KUKA KRL program: MyProgram_312().src

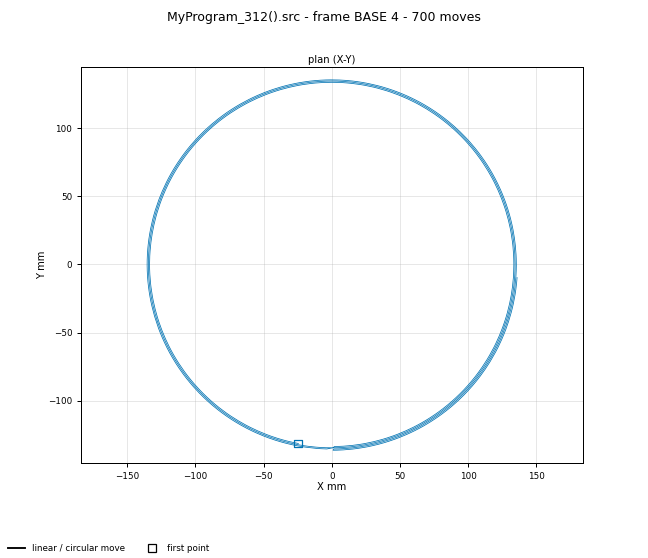
[picture p0: tool path of MyProgram_312().src in frame BASE 4, 700 of 700 moves have a stored position in this frame; points joined in program order, loops and branches not executed]
&ACCESS RVP
&REL 1
&PARAM TEMPLATE = C:\KRC\Roboter\Template\vorgabe
&PARAM EDITMASK = *
DEF MyProgram_312()
; ---- Setting reference (Base) ----
$BASE = BASE_DATA[4]

; --------------------------
; ---- Setting tool (TCP) ----
$TOOL = TOOL_DATA[3]
; --------------------------

$VEL.CP = VEL_APROX_PRINT
Startdeposition()
$VEL.CP = VEL_PRINT
LIN {X -24.4618,Y -131.3769,Z 183,A -96.3174,B 4.4526,C 0.3571,E1 4.4393,E2 188.8666} C_DIS
LIN {X -27.6736,Y -130.7376,Z 183,A -97.6133,B 4.4528,C 0.3555,E1 4.4357,E2 190.1492} C_DIS
LIN {X -30.5793,Y -130.0897,Z 183,A -99.1035,B 4.4527,C 0.3569,E1 4.4316,E2 191.6668} C_DIS
LIN {X -33.6463,Y -129.3306,Z 183,A -100.4108,B 4.4527,C 0.3557,E1 4.4281,E2 192.9686} C_DIS
LIN {X -36.9217,Y -128.4331,Z 183,A -101.7714,B 4.4529,C 0.3539,E1 4.4245,E2 194.3175} C_DIS
LIN {X -40.1243,Y -127.4684,Z 183,A -103.4209,B 4.4529,C 0.3548,E1 4.42,E2 195.9945} C_DIS
LIN {X -44.4742,Y -126.0175,Z 183,A -105.417,B 4.4529,C 0.3535,E1 4.4147,E2 197.9948} C_DIS
LIN {X -48.1013,Y -124.6763,Z 183,A -106.9374,B 4.4531,C 0.3508,E1 4.4108,E2 199.4981} C_DIS
LIN {X -51.1439,Y -123.4595,Z 183,A -108.3574,B 4.4532,C 0.3496,E1 4.4071,E2 200.9202} C_DIS
LIN {X -54.1545,Y -122.1691,Z 183,A -109.7774,B 4.4533,C 0.3483,E1 4.4034,E2 202.3424} C_DIS
LIN {X -57.1353,Y -120.804,Z 183,A -111.0888,B 4.4535,C 0.346,E1 4.4002,E2 203.6421} C_DIS
LIN {X -59.7984,Y -119.5095,Z 183,A -112.49,B 4.4535,C 0.3457,E1 4.3966,E2 205.0601} C_DIS
LIN {X -62.9972,Y -117.8548,Z 183,A -113.9682,B 4.4537,C 0.3433,E1 4.393,E2 206.5301} C_DIS
LIN {X -65.8824,Y -116.2669,Z 183,A -115.4343,B 4.4538,C 0.3419,E1 4.3894,E2 208.0031} C_DIS
LIN {X -68.4366,Y -114.7813,Z 183,A -116.7737,B 4.4539,C 0.3409,E1 4.3861,E2 209.3516} C_DIS
LIN {X -71.2324,Y -113.0676,Z 183,A -118.2015,B 4.454,C 0.3391,E1 4.3827,E2 210.7822} C_DIS
LIN {X -73.9824,Y -111.2879,Z 183,A -119.6266,B 4.4542,C 0.3372,E1 4.3794,E2 212.2099} C_DIS
LIN {X -76.9449,Y -109.2603,Z 183,A -121.1955,B 4.4543,C 0.3351,E1 4.3758,E2 213.7824} C_DIS
LIN {X -79.5983,Y -107.3429,Z 183,A -122.6255,B 4.4545,C 0.3331,E1 4.3725,E2 215.2157} C_DIS
LIN {X -82.0022,Y -105.5177,Z 183,A -123.9905,B 4.4546,C 0.3316,E1 4.3695,E2 216.5895} C_DIS
LIN {X -85.2897,Y -102.8786,Z 183,A -125.8423,B 4.4548,C 0.3288,E1 4.3655,E2 218.4467} C_DIS
LIN {X -88.5217,Y -100.1111,Z 183,A -127.6554,B 4.455,C 0.3255,E1 4.3617,E2 220.2581} C_DIS
LIN {X -91.4468,Y -97.447,Z 183,A -129.5287,B 4.4552,C 0.3237,E1 4.3578,E2 222.1532} C_DIS
LIN {X -94.4975,Y -94.4919,Z 183,A -131.3923,B 4.4554,C 0.3206,E1 4.354,E2 224.0218} C_DIS
LIN {X -97.453,Y -91.4405,Z 183,A -133.251,B 4.4556,C 0.3173,E1 4.3505,E2 225.8848} C_DIS
LIN {X -100.5505,Y -88.0225,Z 183,A -135.1692,B 4.456,C 0.3128,E1 4.3469,E2 227.7951} C_DIS
LIN {X -103.0201,Y -85.1187,Z 183,A -136.9276,B 4.4561,C 0.3102,E1 4.3437,E2 229.5685} C_DIS
LIN {X -105.8538,Y -81.5686,Z 183,A -138.9198,B 4.4564,C 0.3063,E1 4.3403,E2 231.5658} C_DIS
LIN {X -108.1186,Y -78.5411,Z 183,A -140.4676,B 4.4567,C 0.3022,E1 4.3377,E2 233.1039} C_DIS
LIN {X -110.3763,Y -75.336,Z 183,A -142.1523,B 4.4569,C 0.2984,E1 4.335,E2 234.7885} C_DIS
LIN {X -112.0187,Y -72.8707,Z 183,A -143.499,B 4.4571,C 0.296,E1 4.333,E2 236.1443} C_DIS
LIN {X -113.9347,Y -69.8371,Z 183,A -145.1995,B 4.4573,C 0.2935,E1 4.3304,E2 237.8643} C_DIS
LIN {X -116.1262,Y -66.1289,Z 183,A -146.9827,B 4.4576,C 0.2887,E1 4.3279,E2 239.6389} C_DIS
LIN {X -117.7075,Y -63.2714,Z 183,A -148.4758,B 4.4578,C 0.2859,E1 4.3259,E2 241.1429} C_DIS
LIN {X -119.36,Y -60.0943,Z 183,A -150.0116,B 4.458,C 0.2821,E1 4.324,E2 242.6781} C_DIS
LIN {X -120.8057,Y -57.1318,Z 183,A -151.4345,B 4.4582,C 0.2786,E1 4.3222,E2 244.1015} C_DIS
LIN {X -122.0437,Y -54.4348,Z 183,A -152.7707,B 4.4584,C 0.2757,E1 4.3207,E2 245.4449} C_DIS
LIN {X -123.341,Y -51.4275,Z 183,A -154.2178,B 4.4586,C 0.2724,E1 4.3191,E2 246.8967} C_DIS
LIN {X -124.5655,Y -48.3864,Z 183,A -155.6725,B 4.4588,C 0.2691,E1 4.3176,E2 248.3567} C_DIS
LIN {X -125.7252,Y -45.2879,Z 183,A -157.1775,B 4.459,C 0.2659,E1 4.3161,E2 249.8717} C_DIS
LIN {X -126.7947,Y -42.2009,Z 183,A -158.573,B 4.4592,C 0.2621,E1 4.3149,E2 251.2657} C_DIS
LIN {X -127.8799,Y -38.79,Z 183,A -160.1562,B 4.4594,C 0.2583,E1 4.3136,E2 252.8541} C_DIS
LIN {X -128.7913,Y -35.648,Z 183,A -161.6028,B 4.4596,C 0.2548,E1 4.3125,E2 254.3053} C_DIS
LIN {X -129.5522,Y -32.7733,Z 183,A -162.921,B 4.4598,C 0.2516,E1 4.3115,E2 255.628} C_DIS
LIN {X -130.3865,Y -29.2822,Z 183,A -164.5048,B 4.46,C 0.2477,E1 4.3105,E2 257.2165} C_DIS
LIN {X -131.0037,Y -26.3814,Z 183,A -165.8204,B 4.4602,C 0.2445,E1 4.3098,E2 258.5366} C_DIS
LIN {X -131.6133,Y -23.151,Z 183,A -167.2969,B 4.4604,C 0.241,E1 4.309,E2 260.0204} C_DIS
LIN {X -132.1888,Y -19.6089,Z 183,A -168.8833,B 4.4606,C 0.237,E1 4.3084,E2 261.6117} C_DIS
LIN {X -132.5916,Y -16.6691,Z 183,A -170.1742,B 4.4608,C 0.2335,E1 4.3079,E2 262.904} C_DIS
LIN {X -132.9599,Y -13.4162,Z 183,A -171.6515,B 4.461,C 0.2301,E1 4.3074,E2 264.3894} C_DIS
LIN {X -133.2513,Y -10.1075,Z 183,A -173.1085,B 4.4612,C 0.2263,E1 4.3071,E2 265.8494} C_DIS
LIN {X -133.4392,Y -7.2234,Z 183,A -174.5356,B 4.4612,C 0.2239,E1 4.3069,E2 267.2986} C_DIS
LIN {X -133.5854,Y -3.5914,Z 183,A -175.9912,B 4.4615,C 0.2189,E1 4.3067,E2 268.7405} C_DIS
LIN {X -133.6373,Y -0.0053,Z 183,A -177.6118,B 4.4617,C 0.2151,E1 4.3067,E2 270.3702} C_DIS
LIN {X -133.5942,Y 3.2729,Z 183,A -179.0575,B 4.4619,C 0.2113,E1 4.3067,E2 271.8197} C_DIS
LIN {X -133.4881,Y 6.2497,Z 183,A 179.6921,B 4.4621,C 0.2075,E1 4.3069,E2 273.0658} C_DIS
LIN {X -133.2715,Y 9.8307,Z 183,A 178.1093,B 4.4623,C 0.2035,E1 4.3072,E2 274.6529} C_DIS
LIN {X -132.9908,Y 13.0943,Z 183,A 176.6053,B 4.4624,C 0.2001,E1 4.3076,E2 276.1679} C_DIS
LIN {X -132.6304,Y 16.3508,Z 183,A 175.1564,B 4.4626,C 0.1964,E1 4.3081,E2 277.6211} C_DIS
LIN {X -132.2328,Y 19.3008,Z 183,A 173.8334,B 4.4627,C 0.1931,E1 4.3086,E2 278.9488} C_DIS
LIN {X -131.7203,Y 22.5377,Z 183,A 172.2597,B 4.4629,C 0.1903,E1 4.3093,E2 280.5417} C_DIS
LIN {X -131.0418,Y 26.1939,Z 183,A 170.7351,B 4.4631,C 0.1854,E1 4.3101,E2 282.0567} C_DIS
LIN {X -130.4381,Y 29.0563,Z 183,A 169.4367,B 4.4631,C 0.1822,E1 4.3109,E2 283.3594} C_DIS
LIN {X -129.7231,Y 32.0999,Z 183,A 168.0142,B 4.4633,C 0.179,E1 4.3118,E2 284.7907} C_DIS
LIN {X -128.8826,Y 35.3214,Z 183,A 166.5564,B 4.4635,C 0.1753,E1 4.3129,E2 286.2511} C_DIS
LIN {X -127.9681,Y 38.5018,Z 183,A 165.1078,B 4.4636,C 0.1716,E1 4.314,E2 287.7021} C_DIS
LIN {X -126.8894,Y 41.9166,Z 183,A 163.5207,B 4.4638,C 0.1678,E1 4.3154,E2 289.2941} C_DIS
LIN {X -125.9257,Y 44.7317,Z 183,A 162.1162,B 4.4638,C 0.1652,E1 4.3167,E2 290.7129} C_DIS
LIN {X -124.6793,Y 48.0938,Z 183,A 160.6227,B 4.464,C 0.1609,E1 4.3182,E2 292.2} C_DIS
LIN {X -123.4628,Y 51.1359,Z 183,A 159.1751,B 4.4641,C 0.1575,E1 4.3197,E2 293.6515} C_DIS
LIN {X -122.046,Y 54.4295,Z 183,A 157.5018,B 4.4642,C 0.1543,E1 4.3216,E2 295.3398} C_DIS
LIN {X -120.2321,Y 58.3325,Z 183,A 155.681,B 4.4644,C 0.1495,E1 4.3237,E2 297.1562} C_DIS
LIN {X -118.757,Y 61.2788,Z 183,A 154.1805,B 4.4645,C 0.1465,E1 4.3257,E2 298.666} C_DIS
LIN {X -117.0718,Y 64.4409,Z 183,A 152.6549,B 4.4646,C 0.1426,E1 4.3277,E2 300.189} C_DIS
LIN {X -115.4572,Y 67.2912,Z 183,A 151.1996,B 4.4647,C 0.1395,E1 4.3297,E2 301.6493} C_DIS
LIN {X -113.3865,Y 70.7237,Z 183,A 149.3133,B 4.4648,C 0.1365,E1 4.3325,E2 303.554} C_DIS
LIN {X -111.2723,Y 74.0057,Z 183,A 147.7225,B 4.465,C 0.1319,E1 4.3349,E2 305.1336} C_DIS
LIN {X -109.2524,Y 76.9562,Z 183,A 146.2239,B 4.465,C 0.1282,E1 4.3373,E2 306.6268} C_DIS
LIN {X -107.3357,Y 79.608,Z 183,A 144.7072,B 4.4651,C 0.1257,E1 4.3398,E2 308.1559} C_DIS
LIN {X -105.2691,Y 82.3214,Z 183,A 143.0587,B 4.4651,C 0.1238,E1 4.3427,E2 309.8253} C_DIS
LIN {X -102.6063,Y 85.6177,Z 183,A 141.2079,B 4.4653,C 0.12,E1 4.3459,E2 311.6786} C_DIS
LIN {X -99.6528,Y 89.0374,Z 183,A 139.3277,B 4.4654,C 0.1156,E1 4.3494,E2 313.5505} C_DIS
LIN {X -96.9083,Y 92.0178,Z 183,A 137.5407,B 4.4654,C 0.1123,E1 4.3528,E2 315.3419} C_DIS
LIN {X -94.0835,Y 94.9033,Z 183,A 135.7785,B 4.4656,C 0.1091,E1 4.3563,E2 317.1064} C_DIS
LIN {X -91.1824,Y 97.694,Z 183,A 133.9223,B 4.4656,C 0.1067,E1 4.3601,E2 318.9766} C_DIS
LIN {X -87.725,Y 100.8101,Z 183,A 131.8888,B 4.4657,C 0.1033,E1 4.3643,E2 321.0129} C_DIS
LIN {X -84.7137,Y 103.3535,Z 183,A 130.2415,B 4.4657,C 0.1,E1 4.3678,E2 322.6538} C_DIS
LIN {X -81.5394,Y 105.8765,Z 183,A 128.3316,B 4.4658,C 0.0983,E1 4.3721,E2 324.5826} C_DIS
LIN {X -77.7949,Y 108.6567,Z 183,A 126.326,B 4.4658,C 0.0951,E1 4.3766,E2 326.5874} C_DIS
LIN {X -74.2299,Y 111.1226,Z 183,A 124.567,B 4.466,C 0.0914,E1 4.3806,E2 328.3333} C_DIS
LIN {X -71.4844,Y 112.9086,Z 183,A 123.1409,B 4.466,C 0.0895,E1 4.384,E2 329.7609} C_DIS
LIN {X -68.6974,Y 114.6259,Z 183,A 121.7158,B 4.466,C 0.0877,E1 4.3874,E2 331.1875} C_DIS
LIN {X -66.1393,Y 116.1203,Z 183,A 120.419,B 4.466,C 0.0861,E1 4.3905,E2 332.4866} C_DIS
LIN {X -63.2763,Y 117.7049,Z 183,A 118.9475,B 4.466,C 0.0848,E1 4.3942,E2 333.965} C_DIS
LIN {X -60.0793,Y 119.3676,Z 183,A 117.4211,B 4.4661,C 0.0827,E1 4.398,E2 335.4882} C_DIS
LIN {X -57.1341,Y 120.8046,Z 183,A 116.0284,B 4.4661,C 0.081,E1 4.4015,E2 336.8784} C_DIS
LIN {X -54.4385,Y 122.042,Z 183,A 114.7042,B 4.4661,C 0.08,E1 4.4048,E2 338.2079} C_DIS
LIN {X -51.3816,Y 123.3602,Z 183,A 113.2716,B 4.4662,C 0.0785,E1 4.4085,E2 339.6402} C_DIS
LIN {X -48.3609,Y 124.5754,Z 183,A 111.8116,B 4.4662,C 0.0777,E1 4.4123,E2 341.1067} C_DIS
LIN {X -44.3513,Y 126.0601,Z 183,A 109.8542,B 4.4662,C 0.077,E1 4.4175,E2 343.0776} C_DIS
LIN {X -40.6686,Y 127.2945,Z 183,A 108.274,B 4.4662,C 0.075,E1 4.4217,E2 344.6467} C_DIS
LIN {X -37.2161,Y 128.3468,Z 183,A 106.7647,B 4.4662,C 0.0735,E1 4.4257,E2 346.1506} C_DIS
LIN {X -34.0571,Y 129.2212,Z 183,A 105.3495,B 4.4663,C 0.0726,E1 4.4295,E2 347.5661} C_DIS
LIN {X -31.1805,Y 129.9448,Z 183,A 104.0275,B 4.4663,C 0.0722,E1 4.4331,E2 348.8932} C_DIS
LIN {X -27.6666,Y 130.7391,Z 183,A 102.54,B 4.4663,C 0.0709,E1 4.4372,E2 350.3732} C_DIS
LIN {X -24.7582,Y 131.3203,Z 183,A 101.2384,B 4.4663,C 0.0706,E1 4.4407,E2 351.6775} C_DIS
LIN {X -21.225,Y 131.9393,Z 183,A 99.6763,B 4.4663,C 0.0702,E1 4.4451,E2 353.2417} C_DIS
LIN {X -17.9865,Y 132.4189,Z 183,A 98.3524,B 4.4663,C 0.069,E1 4.4487,E2 354.5555} C_DIS
LIN {X -15.0176,Y 132.7889,Z 183,A 96.9769,B 4.4663,C 0.0695,E1 4.4525,E2 355.9412} C_DIS
LIN {X -11.7619,Y 133.1159,Z 183,A 95.3739,B 4.4663,C 0.071,E1 4.4571,E2 357.567} C_DIS
LIN {X -6.5548,Y 133.4728,Z 183,A 93.3522,B 4.4663,C 0.0688,E1 4.4626,E2 359.5623} C_DIS
LIN {X -3.6395,Y 133.584,Z 183,A 92.0894,B 4.4663,C 0.0688,E1 4.4661,E2 360.8259} C_DIS
LIN {X -0.2953,Y 133.634,Z 183,A 90.6127,B 4.4663,C 0.0693,E1 4.4703,E2 362.3069} C_DIS
LIN {X 3.2877,Y 133.5938,Z 183,A 89.0043,B 4.4663,C 0.0702,E1 4.4748,E2 363.9232} C_DIS
LIN {X 7.8852,Y 133.4011,Z 183,A 87.0874,B 4.4663,C 0.07,E1 4.4801,E2 365.8327} C_DIS
LIN {X 11.1511,Y 133.1675,Z 183,A 85.7051,B 4.4663,C 0.0702,E1 4.484,E2 367.2119} C_DIS
LIN {X 14.7355,Y 132.8193,Z 183,A 84.2303,B 4.4663,C 0.0702,E1 4.488,E2 368.6781} C_DIS
LIN {X 17.9896,Y 132.4185,Z 183,A 82.8458,B 4.4663,C 0.0705,E1 4.4919,E2 370.0596} C_DIS
LIN {X 20.9212,Y 131.9864,Z 183,A 81.5656,B 4.4663,C 0.0712,E1 4.4954,E2 371.3405} C_DIS
LIN {X 24.4587,Y 131.3775,Z 183,A 80.0946,B 4.4663,C 0.0714,E1 4.4994,E2 372.8031} C_DIS
LIN {X 27.6823,Y 130.7357,Z 183,A 78.7373,B 4.4663,C 0.0718,E1 4.5031,E2 374.1539} C_DIS
LIN {X 30.4017,Y 130.1308,Z 183,A 77.3268,B 4.4663,C 0.0748,E1 4.507,E2 375.5895} C_DIS
LIN {X 33.7569,Y 129.3012,Z 183,A 76.0205,B 4.4663,C 0.0742,E1 4.5105,E2 376.8748} C_DIS
LIN {X 36.9909,Y 128.4128,Z 183,A 74.5572,B 4.4663,C 0.0756,E1 4.5145,E2 378.3407} C_DIS
LIN {X 40.0825,Y 127.4817,Z 183,A 73.2386,B 4.4663,C 0.0762,E1 4.518,E2 379.6513} C_DIS
LIN {X 43.4821,Y 126.3615,Z 183,A 71.7611,B 4.4663,C 0.077,E1 4.5219,E2 381.1217} C_DIS
LIN {X 46.5669,Y 125.2575,Z 183,A 70.2745,B 4.4662,C 0.0793,E1 4.5258,E2 382.6177} C_DIS
LIN {X 49.6229,Y 124.0786,Z 183,A 68.8881,B 4.4662,C 0.0807,E1 4.5294,E2 384.0018} C_DIS
LIN {X 52.6515,Y 122.8242,Z 183,A 67.5024,B 4.4662,C 0.0821,E1 4.533,E2 385.385} C_DIS
LIN {X 55.6459,Y 121.4971,Z 183,A 66.1184,B 4.4662,C 0.0836,E1 4.5365,E2 386.7664} C_DIS
LIN {X 58.3271,Y 120.2347,Z 183,A 64.854,B 4.4661,C 0.0851,E1 4.5397,E2 388.0301} C_DIS
LIN {X 61.2694,Y 118.7618,Z 183,A 63.4176,B 4.4661,C 0.0873,E1 4.5432,E2 389.4694} C_DIS
LIN {X 64.451,Y 117.0662,Z 183,A 61.9594,B 4.4661,C 0.0885,E1 4.5468,E2 390.9172} C_DIS
LIN {X 67.2814,Y 115.4629,Z 183,A 60.6146,B 4.466,C 0.09,E1 4.55,E2 392.256} C_DIS
LIN {X 69.8405,Y 113.9326,Z 183,A 59.3243,B 4.466,C 0.0921,E1 4.5531,E2 393.5477} C_DIS
LIN {X 72.6093,Y 112.1884,Z 183,A 57.9479,B 4.466,C 0.094,E1 4.5564,E2 394.9209} C_DIS
LIN {X 75.3362,Y 110.3761,Z 183,A 56.497,B 4.4659,C 0.0968,E1 4.5597,E2 396.3775} C_DIS
LIN {X 78.8584,Y 107.8878,Z 183,A 54.6474,B 4.4658,C 0.0999,E1 4.5639,E2 398.2273} C_DIS
LIN {X 82.219,Y 105.3495,Z 183,A 52.8465,B 4.4658,C 0.103,E1 4.5679,E2 400.0277} C_DIS
LIN {X 85.5311,Y 102.6786,Z 183,A 51.0551,B 4.4656,C 0.106,E1 4.5718,E2 401.8155} C_DIS
LIN {X 89.0339,Y 99.6559,Z 183,A 49.2239,B 4.4656,C 0.108,E1 4.5756,E2 403.6287} C_DIS
LIN {X 92.0406,Y 96.8866,Z 183,A 47.5065,B 4.4656,C 0.1111,E1 4.5791,E2 405.3422} C_DIS
LIN {X 94.9606,Y 94.0258,Z 183,A 45.7768,B 4.4654,C 0.1144,E1 4.5825,E2 407.0695} C_DIS
LIN {X 97.9101,Y 90.9503,Z 183,A 43.9171,B 4.4654,C 0.1185,E1 4.5861,E2 408.9334} C_DIS
LIN {X 100.6522,Y 87.906,Z 183,A 42.2099,B 4.4652,C 0.1217,E1 4.5893,E2 410.6351} C_DIS
LIN {X 103.6922,Y 84.2992,Z 183,A 40.2826,B 4.4652,C 0.1251,E1 4.5927,E2 412.5517} C_DIS
LIN {X 106.3516,Y 80.9184,Z 183,A 38.4212,B 4.465,C 0.1294,E1 4.5959,E2 414.4156} C_DIS
LIN {X 109.0871,Y 77.1904,Z 183,A 36.6295,B 4.465,C 0.1318,E1 4.5988,E2 416.185} C_DIS
LIN {X 111.1167,Y 74.2389,Z 183,A 35.131,B 4.4649,C 0.1349,E1 4.6011,E2 417.6796} C_DIS
LIN {X 112.9026,Y 71.4939,Z 183,A 33.8268,B 4.4648,C 0.1371,E1 4.6031,E2 418.9722} C_DIS
LIN {X 114.6206,Y 68.7063,Z 183,A 32.4025,B 4.4647,C 0.1408,E1 4.6051,E2 420.3996} C_DIS
LIN {X 116.0831,Y 66.2045,Z 183,A 31.1744,B 4.4646,C 0.1436,E1 4.6068,E2 421.6264} C_DIS
LIN {X 117.707,Y 63.2723,Z 183,A 29.7413,B 4.4645,C 0.1472,E1 4.6088,E2 423.0595} C_DIS
LIN {X 119.3644,Y 60.0857,Z 183,A 28.2876,B 4.4644,C 0.15,E1 4.6106,E2 424.5035} C_DIS
LIN {X 120.8068,Y 57.1295,Z 183,A 26.9475,B 4.4643,C 0.1528,E1 4.6122,E2 425.8357} C_DIS
LIN {X 122.0435,Y 54.4353,Z 183,A 25.689,B 4.4642,C 0.1559,E1 4.6137,E2 427.0933} C_DIS
LIN {X 123.3407,Y 51.4282,Z 183,A 24.3261,B 4.4641,C 0.1591,E1 4.6151,E2 428.4518} C_DIS
LIN {X 124.5639,Y 48.3904,Z 183,A 22.9635,B 4.464,C 0.1623,E1 4.6165,E2 429.8101} C_DIS
LIN {X 125.7122,Y 45.3239,Z 183,A 21.5517,B 4.4638,C 0.1661,E1 4.6179,E2 431.2236} C_DIS
LIN {X 126.7222,Y 42.4188,Z 183,A 20.2778,B 4.4638,C 0.1691,E1 4.619,E2 432.4927} C_DIS
LIN {X 127.7915,Y 39.0787,Z 183,A 18.818,B 4.4636,C 0.1726,E1 4.6202,E2 433.9481} C_DIS
LIN {X 128.7935,Y 35.6399,Z 183,A 17.3754,B 4.4635,C 0.1757,E1 4.6213,E2 435.3803} C_DIS
LIN {X 129.563,Y 32.7306,Z 183,A 16.1299,B 4.4633,C 0.1786,E1 4.6222,E2 436.621} C_DIS
LIN {X 130.3866,Y 29.2818,Z 183,A 14.6546,B 4.4632,C 0.1823,E1 4.6231,E2 438.0917} C_DIS
LIN {X 131.0067,Y 26.3666,Z 183,A 13.4138,B 4.4631,C 0.1854,E1 4.6238,E2 439.3288} C_DIS
LIN {X 131.6138,Y 23.148,Z 183,A 12.0336,B 4.4629,C 0.189,E1 4.6245,E2 440.7069} C_DIS
LIN {X 132.1889,Y 19.608,Z 183,A 10.5465,B 4.4628,C 0.1926,E1 4.6252,E2 442.1889} C_DIS
LIN {X 132.5912,Y 16.6722,Z 183,A 9.3378,B 4.4626,C 0.1954,E1 4.6256,E2 443.3909} C_DIS
LIN {X 132.9609,Y 13.4062,Z 183,A 7.9487,B 4.4625,C 0.1992,E1 4.626,E2 444.7784} C_DIS
LIN {X 133.272,Y 9.8231,Z 183,A 6.5357,B 4.4623,C 0.2019,E1 4.6263,E2 446.1766} C_DIS
LIN {X 133.4694,Y 6.6226,Z 183,A 5.1329,B 4.4622,C 0.2061,E1 4.6266,E2 447.5838} C_DIS
LIN {X 133.5853,Y 3.594,Z 183,A 3.8849,B 4.462,C 0.2092,E1 4.6266,E2 448.8263} C_DIS
LIN {X 133.6372,Y -0.023,Z 183,A 2.3601,B 4.4618,C 0.2132,E1 4.6267,E2 450.3491} C_DIS
LIN {X 133.5938,Y -3.2887,Z 183,A 1.0075,B 4.4617,C 0.2166,E1 4.6267,E2 451.6968} C_DIS
LIN {X 133.488,Y -6.2516,Z 183,A -0.224,B 4.4615,C 0.2197,E1 4.6265,E2 452.9244} C_DIS
LIN {X 133.2715,Y -9.8297,Z 183,A -1.6445,B 4.4614,C 0.2226,E1 4.6262,E2 454.3317} C_DIS
LIN {X 132.991,Y -13.0926,Z 183,A -3.0547,B 4.4612,C 0.2266,E1 4.6259,E2 455.7437} C_DIS
LIN {X 132.6287,Y -16.365,Z 183,A -4.4179,B 4.461,C 0.23,E1 4.6254,E2 457.102} C_DIS
LIN {X 132.2326,Y -19.3022,Z 183,A -5.6531,B 4.4608,C 0.2331,E1 4.625,E2 458.3338} C_DIS
LIN {X 131.72,Y -22.5395,Z 183,A -7.0691,B 4.4606,C 0.2372,E1 4.6243,E2 459.7523} C_DIS
LIN {X 131.0676,Y -26.0672,Z 183,A -8.5189,B 4.4604,C 0.2404,E1 4.6236,E2 461.1923} C_DIS
LIN {X 130.4587,Y -28.9656,Z 183,A -9.7453,B 4.4603,C 0.2434,E1 4.6228,E2 462.4145} C_DIS
LIN {X 129.6388,Y -32.432,Z 183,A -11.1368,B 4.4601,C 0.2459,E1 4.6219,E2 463.7902} C_DIS
LIN {X 128.8766,Y -35.3426,Z 183,A -12.4766,B 4.4599,C 0.2501,E1 4.621,E2 465.1373} C_DIS
LIN {X 127.972,Y -38.489,Z 183,A -13.8372,B 4.4597,C 0.2534,E1 4.6199,E2 466.4937} C_DIS
LIN {X 126.7798,Y -42.2458,Z 183,A -15.5567,B 4.4594,C 0.2583,E1 4.6184,E2 468.2182} C_DIS
LIN {X 125.258,Y -46.5656,Z 183,A -17.2326,B 4.4594,C 0.26,E1 4.6169,E2 469.86} C_DIS
LIN {X 124.0822,Y -49.6139,Z 183,A -18.7362,B 4.459,C 0.265,E1 4.6153,E2 471.3776} C_DIS
LIN {X 122.8228,Y -52.6548,Z 183,A -20.1062,B 4.4589,C 0.2683,E1 4.6138,E2 472.7437} C_DIS
LIN {X 121.4946,Y -55.6513,Z 183,A -21.47,B 4.4587,C 0.2714,E1 4.6123,E2 474.1035} C_DIS
LIN {X 120.2321,Y -58.3325,Z 183,A -22.713,B 4.4585,C 0.2744,E1 4.6108,E2 475.3442} C_DIS
LIN {X 118.7502,Y -61.2922,Z 183,A -24.1373,B 4.4583,C 0.2781,E1 4.609,E2 476.7703} C_DIS
LIN {X 117.0664,Y -64.4506,Z 183,A -25.573,B 4.4581,C 0.2807,E1 4.6071,E2 478.195} C_DIS
LIN {X 115.801,Y -66.6973,Z 183,A -26.7315,B 4.4579,C 0.2842,E1 4.6055,E2 479.3611} C_DIS
LIN {X 113.9338,Y -69.8385,Z 183,A -28.1752,B 4.4577,C 0.2865,E1 4.6034,E2 480.7907} C_DIS
LIN {X 112.1907,Y -72.6058,Z 183,A -29.5368,B 4.4575,C 0.2894,E1 4.6014,E2 482.1484} C_DIS
LIN {X 110.3815,Y -75.3285,Z 183,A -31.0271,B 4.4572,C 0.2939,E1 4.599,E2 483.651} C_DIS
LIN {X 107.7956,Y -78.984,Z 183,A -32.9007,B 4.457,C 0.2978,E1 4.596,E2 485.5205} C_DIS
LIN {X 105.3479,Y -82.2211,Z 183,A -34.6049,B 4.4567,C 0.3014,E1 4.5931,E2 487.2217} C_DIS
LIN {X 102.6786,Y -85.5311,Z 183,A -36.382,B 4.4565,C 0.305,E1 4.5899,E2 488.9946} C_DIS
LIN {X 99.6714,Y -89.0166,Z 183,A -38.204,B 4.4563,C 0.3075,E1 4.5866,E2 490.7993} C_DIS
LIN {X 96.8883,Y -92.0388,Z 183,A -39.9265,B 4.4561,C 0.3108,E1 4.5833,E2 492.5184} C_DIS
LIN {X 94.0228,Y -94.9636,Z 183,A -41.6547,B 4.4559,C 0.3141,E1 4.5799,E2 494.2446} C_DIS
LIN {X 90.9533,Y -97.9073,Z 183,A -43.5139,B 4.4556,C 0.3182,E1 4.5762,E2 496.1098} C_DIS
LIN {X 87.9022,Y -100.6555,Z 183,A -45.2259,B 4.4554,C 0.3211,E1 4.5726,E2 497.8172} C_DIS
LIN {X 84.7758,Y -103.3028,Z 183,A -46.8635,B 4.4552,C 0.323,E1 4.5691,E2 499.4412} C_DIS
LIN {X 81.57,Y -105.8527,Z 183,A -48.657,B 4.455,C 0.3267,E1 4.5651,E2 501.2409} C_DIS
LIN {X 78.5425,Y -108.1177,Z 183,A -50.1367,B 4.4549,C 0.3279,E1 4.5619,E2 502.7041} C_DIS
LIN {X 75.8581,Y -110.018,Z 183,A -51.6127,B 4.4546,C 0.3311,E1 4.5584,E2 504.1896} C_DIS
LIN {X 72.8032,Y -112.0626,Z 183,A -53.0653,B 4.4546,C 0.3323,E1 4.5551,E2 505.6277} C_DIS
LIN {X 70.0612,Y -113.7972,Z 183,A -54.5614,B 4.4543,C 0.3357,E1 4.5515,E2 507.1382} C_DIS
LIN {X 66.125,Y -116.1285,Z 183,A -56.3627,B 4.4543,C 0.3369,E1 4.5472,E2 508.9209} C_DIS
LIN {X 63.2772,Y -117.7044,Z 183,A -57.7862,B 4.454,C 0.3392,E1 4.5437,E2 510.3489} C_DIS
LIN {X 60.075,Y -119.3698,Z 183,A -59.2655,B 4.454,C 0.3406,E1 4.54,E2 511.8208} C_DIS
LIN {X 57.1312,Y -120.806,Z 183,A -60.6187,B 4.4538,C 0.3419,E1 4.5367,E2 513.1685} C_DIS
LIN {X 54.4362,Y -122.0431,Z 183,A -61.8542,B 4.4538,C 0.3432,E1 4.5335,E2 514.4003} C_DIS
LIN {X 51.4282,Y -123.3408,Z 183,A -63.2809,B 4.4536,C 0.3451,E1 4.5298,E2 515.8309} C_DIS
LIN {X 48.3909,Y -124.5638,Z 183,A -64.6664,B 4.4535,C 0.3466,E1 4.5262,E2 517.215} C_DIS
LIN {X 45.0269,Y -125.8193,Z 183,A -66.2957,B 4.4533,C 0.3492,E1 4.5219,E2 518.8567} C_DIS
LIN {X 40.6558,Y -127.2986,Z 183,A -68.1923,B 4.4532,C 0.3504,E1 4.5169,E2 520.7443} C_DIS
LIN {X 37.2146,Y -128.3473,Z 183,A -69.6673,B 4.4532,C 0.3511,E1 4.513,E2 522.2118} C_DIS
LIN {X 34.0546,Y -129.2218,Z 183,A -71.058,B 4.453,C 0.3521,E1 4.5093,E2 523.6015} C_DIS
LIN {X 31.1781,Y -129.9454,Z 183,A -72.3579,B 4.453,C 0.3534,E1 4.5057,E2 524.9058} C_DIS
LIN {X 27.6802,Y -130.7362,Z 183,A -73.8168,B 4.4529,C 0.3537,E1 4.5018,E2 526.3557} C_DIS
LIN {X 24.7521,Y -131.3214,Z 183,A -75.111,B 4.4529,C 0.3547,E1 4.4982,E2 527.6524} C_DIS
LIN {X 21.2186,Y -131.9404,Z 183,A -76.6564,B 4.4527,C 0.3558,E1 4.4939,E2 529.1997} C_DIS
LIN {X 17.9806,Y -132.4197,Z 183,A -77.9638,B 4.4527,C 0.3555,E1 4.4904,E2 530.4957} C_DIS
LIN {X 15.0397,Y -132.7865,Z 183,A -79.3186,B 4.4527,C 0.357,E1 4.4866,E2 531.8618} C_DIS
LIN {X 11.7495,Y -133.1169,Z 183,A -80.7949,B 4.4525,C 0.3581,E1 4.4824,E2 533.3463} C_DIS
LIN {X 8.4886,Y -133.3639,Z 183,A -82.1732,B 4.4525,C 0.3584,E1 4.4786,E2 534.7223} C_DIS
LIN {X 4.913,Y -133.5436,Z 183,A -83.5921,B 4.4525,C 0.3576,E1 4.4747,E2 536.1273} C_DIS
LIN {X 1.9511,Y -133.6196,Z 183,A -84.8958,B 4.4525,C 0.3582,E1 4.471,E2 537.4359} C_DIS
LIN {X 1.9511,Y -133.6196,Z 183,A -84.8958,B 4.4525,C 0.3582,E1 4.471,E2 537.4359} C_DIS
Enddeposition()
LIN {X 0.9664,Y -134.5293,Z 183,A -85.4371,B 4.4523,C 0.3619,E1 4.4694,E2 538.0245} C_DIS
Startdeposition()
$VEL.CP = VEL_PRINT
LIN {X 4.8735,Y -134.4468,Z 183,A -83.1565,B 4.4528,C 0.3554,E1 4.476,E2 535.6644} C_DIS
LIN {X 7.9763,Y -134.2982,Z 183,A -81.9027,B 4.4528,C 0.3557,E1 4.4795,E2 534.4189} C_DIS
LIN {X 11.9917,Y -134.0007,Z 183,A -79.9135,B 4.453,C 0.3523,E1 4.4851,E2 532.3934} C_DIS
LIN {X 15.1883,Y -133.6765,Z 183,A -78.4718,B 4.4531,C 0.3509,E1 4.4891,E2 530.9415} C_DIS
LIN {X 19.3736,Y -133.1326,Z 183,A -76.8302,B 4.4531,C 0.3516,E1 4.4936,E2 529.319} C_DIS
LIN {X 23.4596,Y -132.4734,Z 183,A -74.9289,B 4.4533,C 0.349,E1 4.4989,E2 527.3988} C_DIS
LIN {X 28.1342,Y -131.56,Z 183,A -73.173,B 4.4532,C 0.3506,E1 4.5036,E2 525.6768} C_DIS
LIN {X 31.0475,Y -130.9037,Z 183,A -71.897,B 4.4532,C 0.3495,E1 4.5071,E2 524.3995} C_DIS
LIN {X 34.6302,Y -130.0008,Z 183,A -70.2736,B 4.4534,C 0.3477,E1 4.5115,E2 522.7686} C_DIS
LIN {X 37.9385,Y -129.0742,Z 183,A -68.7972,B 4.4535,C 0.3462,E1 4.5155,E2 521.2896} C_DIS
LIN {X 41.6664,Y -127.9216,Z 183,A -67.0212,B 4.4537,C 0.3433,E1 4.5203,E2 519.4978} C_DIS
LIN {X 45.6366,Y -126.5572,Z 183,A -65.4296,B 4.4537,C 0.3436,E1 4.5244,E2 517.9302} C_DIS
LIN {X 48.2965,Y -125.5671,Z 183,A -64.2321,B 4.4537,C 0.3424,E1 4.5275,E2 516.7334} C_DIS
LIN {X 51.7502,Y -124.1827,Z 183,A -62.6257,B 4.454,C 0.3402,E1 4.5317,E2 515.1231} C_DIS
LIN {X 54.4348,Y -123.0307,Z 183,A -61.5276,B 4.454,C 0.3403,E1 4.5344,E2 514.0428} C_DIS
LIN {X 57.7495,Y -121.5092,Z 183,A -59.9836,B 4.4541,C 0.3384,E1 4.5384,E2 512.4988} C_DIS
LIN {X 60.3618,Y -120.2349,Z 183,A -58.0717,B 4.4548,C 0.3289,E1 4.5434,E2 510.4991} C_DIS
LIN {X 64.7137,Y -117.95,Z 183,A -56.7807,B 4.4543,C 0.3352,E1 4.5463,E2 509.3101} C_DIS
LIN {X 70.9522,Y -114.3056,Z 183,A -53.1134,B 4.4552,C 0.3235,E1 4.5553,E2 505.5645} C_DIS
LIN {X 74.5125,Y -112.0174,Z 183,A -51.7225,B 4.4551,C 0.3254,E1 4.5584,E2 504.2254} C_DIS
LIN {X 78.0908,Y -109.5528,Z 183,A -49.8996,B 4.4553,C 0.3225,E1 4.5625,E2 502.4045} C_DIS
LIN {X 81.6424,Y -106.9322,Z 183,A -48.0641,B 4.4555,C 0.3197,E1 4.5666,E2 500.5731} C_DIS
LIN {X 85.1096,Y -104.1936,Z 183,A -46.2359,B 4.4557,C 0.3168,E1 4.5706,E2 498.7503} C_DIS
LIN {X 88.5551,Y -101.2816,Z 183,A -44.3601,B 4.4559,C 0.3137,E1 4.5746,E2 496.8787} C_DIS
LIN {X 91.7405,Y -98.4054,Z 183,A -42.5589,B 4.4561,C 0.3104,E1 4.5783,E2 495.0794} C_DIS
LIN {X 94.9711,Y -95.2915,Z 183,A -40.6998,B 4.4564,C 0.307,E1 4.582,E2 493.2255} C_DIS
LIN {X 98.1179,Y -92.0487,Z 183,A -38.825,B 4.4566,C 0.3036,E1 4.5856,E2 491.3554} C_DIS
LIN {X 100.8751,Y -89.0178,Z 183,A -37.1086,B 4.4568,C 0.3001,E1 4.5888,E2 489.6411} C_DIS
LIN {X 103.8278,Y -85.5561,Z 183,A -35.2091,B 4.4571,C 0.2963,E1 4.5922,E2 487.7449} C_DIS
LIN {X 106.5718,Y -82.113,Z 183,A -33.3635,B 4.4574,C 0.2923,E1 4.5953,E2 485.9015} C_DIS
LIN {X 110.7552,Y -76.3763,Z 183,A -30.5358,B 4.4577,C 0.2877,E1 4.5999,E2 483.0963} C_DIS
LIN {X 112.9406,Y -73.1055,Z 183,A -28.822,B 4.4579,C 0.2831,E1 4.6026,E2 481.3761} C_DIS
LIN {X 115.2347,Y -69.4331,Z 183,A -27.0741,B 4.4582,C 0.2798,E1 4.6051,E2 479.6389} C_DIS
LIN {X 117.2445,Y -65.9824,Z 183,A -25.3993,B 4.4584,C 0.2759,E1 4.6074,E2 477.9659} C_DIS
LIN {X 119.9025,Y -61.0148,Z 183,A -23.1494,B 4.4587,C 0.2716,E1 4.6103,E2 475.733} C_DIS
LIN {X 121.1541,Y -58.4928,Z 183,A -21.8356,B 4.4589,C 0.2671,E1 4.6119,E2 474.4037} C_DIS
LIN {X 122.7409,Y -55.0827,Z 183,A -20.5009,B 4.4589,C 0.2663,E1 4.6135,E2 473.1015} C_DIS
LIN {X 123.8711,Y -52.4965,Z 183,A -18.7536,B 4.4596,C 0.2562,E1 4.6154,E2 471.2838} C_DIS
LIN {X 125.4567,Y -48.5807,Z 183,A -17.5005,B 4.4595,C 0.2584,E1 4.6167,E2 470.0987} C_DIS
LIN {X 128.143,Y -40.9733,Z 183,A -14.2084,B 4.4599,C 0.2509,E1 4.6197,E2 466.8221} C_DIS
LIN {X 129.0157,Y -38.1384,Z 183,A -13.0016,B 4.46,C 0.2482,E1 4.6206,E2 465.6214} C_DIS
LIN {X 129.9502,Y -34.82,Z 183,A -11.4613,B 4.4603,C 0.2432,E1 4.6218,E2 464.0708} C_DIS
LIN {X 130.8758,Y -31.1633,Z 183,A -9.83,B 4.4606,C 0.2385,E1 4.6228,E2 462.4351} C_DIS
LIN {X 131.8604,Y -26.6899,Z 183,A -8.0135,B 4.4608,C 0.2348,E1 4.6239,E2 460.634} C_DIS
LIN {X 132.6042,Y -22.7151,Z 183,A -6.4867,B 4.4608,C 0.2325,E1 4.6246,E2 459.1305} C_DIS
LIN {X 133.0757,Y -19.772,Z 183,A -5.0282,B 4.4612,C 0.2264,E1 4.6252,E2 457.6473} C_DIS
LIN {X 133.5433,Y -16.3053,Z 183,A -3.8029,B 4.4612,C 0.2257,E1 4.6257,E2 456.454} C_DIS
LIN {X 134.0237,Y -11.7197,Z 183,A -1.9782,B 4.4614,C 0.2219,E1 4.6262,E2 454.6453} C_DIS
LIN {X 134.2806,Y -8.262,Z 183,A -0.3364,B 4.4617,C 0.2156,E1 4.6265,E2 452.9816} C_DIS
LIN {X 134.4803,Y -3.8222,Z 183,A 1.5169,B 4.462,C 0.2107,E1 4.6267,E2 451.132} C_DIS
LIN {X 134.534,Y 0.666,Z 183,A 3.4741,B 4.4622,C 0.2047,E1 4.6267,E2 449.1677} C_DIS
LIN {X 134.4431,Y 4.9691,Z 183,A 4.9329,B 4.4622,C 0.2043,E1 4.6266,E2 447.7544} C_DIS
LIN {X 134.3323,Y 7.4041,Z 183,A 6.1548,B 4.4625,C 0.199,E1 4.6264,E2 446.5089} C_DIS
LIN {X 134.002,Y 11.9758,Z 183,A 8.1001,B 4.4627,C 0.1936,E1 4.626,E2 444.5631} C_DIS
LIN {X 133.5019,Y 16.6517,Z 183,A 9.9368,B 4.4629,C 0.1901,E1 4.6254,E2 442.7459} C_DIS
LIN {X 132.9672,Y 20.4754,Z 183,A 11.5343,B 4.463,C 0.1861,E1 4.6247,E2 441.1531} C_DIS
LIN {X 132.2732,Y 24.5722,Z 183,A 13.3066,B 4.4632,C 0.1811,E1 4.6239,E2 439.3793} C_DIS
LIN {X 131.5155,Y 28.34,Z 183,A 14.799,B 4.4634,C 0.1784,E1 4.623,E2 437.9039} C_DIS
LIN {X 130.7736,Y 31.5869,Z 183,A 16.1288,B 4.4634,C 0.1756,E1 4.6222,E2 436.5842} C_DIS
LIN {X 130.1412,Y 34.1038,Z 183,A 17.1763,B 4.4636,C 0.1733,E1 4.6215,E2 435.5433} C_DIS
LIN {X 129.2934,Y 37.1898,Z 183,A 18.6769,B 4.4638,C 0.1678,E1 4.6203,E2 434.0249} C_DIS
LIN {X 128.2069,Y 40.7733,Z 183,A 20.1371,B 4.4638,C 0.1652,E1 4.6191,E2 432.5805} C_DIS
LIN {X 126.6453,Y 45.3925,Z 183,A 22.2307,B 4.4641,C 0.1594,E1 4.6172,E2 430.4836} C_DIS
LIN {X 125.1051,Y 49.4852,Z 183,A 24.1109,B 4.4643,C 0.1543,E1 4.6153,E2 428.6003} C_DIS
LIN {X 123.5961,Y 53.1367,Z 183,A 25.4356,B 4.4643,C 0.1543,E1 4.6139,E2 427.319} C_DIS
LIN {X 122.1841,Y 56.3071,Z 183,A 26.8686,B 4.4643,C 0.1511,E1 4.6123,E2 425.8908} C_DIS
LIN {X 120.77,Y 59.2797,Z 183,A 28.3918,B 4.4645,C 0.146,E1 4.6104,E2 424.3522} C_DIS
LIN {X 119.2026,Y 62.3713,Z 183,A 29.779,B 4.4646,C 0.1433,E1 4.6087,E2 422.9752} C_DIS
LIN {X 117.2438,Y 65.9837,Z 183,A 31.5943,B 4.4648,C 0.1382,E1 4.6062,E2 421.1513} C_DIS
LIN {X 115.0468,Y 69.7439,Z 183,A 33.2886,B 4.4648,C 0.1356,E1 4.6038,E2 419.476} C_DIS
LIN {X 113.0482,Y 72.9397,Z 183,A 35.0089,B 4.465,C 0.1304,E1 4.6012,E2 417.7411} C_DIS
LIN {X 110.8627,Y 76.2197,Z 183,A 36.6064,B 4.4651,C 0.1274,E1 4.5987,E2 416.1529} C_DIS
LIN {X 108.2357,Y 79.9066,Z 183,A 38.4693,B 4.4652,C 0.1237,E1 4.5957,E2 414.2974} C_DIS
LIN {X 105.6609,Y 83.2812,Z 183,A 40.1961,B 4.4652,C 0.1206,E1 4.5927,E2 412.5799} C_DIS
LIN {X 103.2828,Y 86.2133,Z 183,A 41.8561,B 4.4654,C 0.1164,E1 4.5898,E2 410.9132} C_DIS
LIN {X 100.2855,Y 89.6815,Z 183,A 43.7111,B 4.4654,C 0.1134,E1 4.5864,E2 409.0696} C_DIS
LIN {X 97.4348,Y 92.771,Z 183,A 45.5237,B 4.4656,C 0.1094,E1 4.5829,E2 407.2539} C_DIS
LIN {X 94.2178,Y 96.0363,Z 183,A 47.3366,B 4.4656,C 0.1071,E1 4.5793,E2 405.4577} C_DIS
LIN {X 90.8324,Y 99.2447,Z 183,A 49.562,B 4.4658,C 0.1004,E1 4.5747,E2 403.2027} C_DIS
LIN {X 88.2437,Y 101.5533,Z 183,A 50.7581,B 4.4658,C 0.1008,E1 4.5723,E2 402.0408} C_DIS
LIN {X 85.0581,Y 104.2357,Z 183,A 52.4739,B 4.4658,C 0.0982,E1 4.5686,E2 400.3317} C_DIS
LIN {X 81.9766,Y 106.6765,Z 183,A 54.1762,B 4.4659,C 0.0949,E1 4.5648,E2 398.626} C_DIS
LIN {X 78.9125,Y 108.9622,Z 183,A 55.7388,B 4.4659,C 0.0929,E1 4.5613,E2 397.0712} C_DIS
LIN {X 75.1503,Y 111.5907,Z 183,A 57.6715,B 4.466,C 0.0899,E1 4.5569,E2 395.1411} C_DIS
LIN {X 71.7434,Y 113.8106,Z 183,A 59.3423,B 4.466,C 0.0879,E1 4.553,E2 393.4777} C_DIS
LIN {X 68.5242,Y 115.7781,Z 183,A 61.0093,B 4.4661,C 0.0848,E1 4.549,E2 391.8034} C_DIS
LIN {X 62.4913,Y 119.1396,Z 183,A 63.8151,B 4.4661,C 0.0822,E1 4.5421,E2 389.0141} C_DIS
LIN {X 58.4184,Y 121.1896,Z 183,A 65.6639,B 4.4661,C 0.0807,E1 4.5375,E2 387.1767} C_DIS
LIN {X 55.3963,Y 122.6007,Z 183,A 67.1687,B 4.4662,C 0.078,E1 4.5337,E2 385.6619} C_DIS
LIN {X 51.9576,Y 124.0961,Z 183,A 68.6192,B 4.4662,C 0.0777,E1 4.53,E2 384.2293} C_DIS
LIN {X 49.4865,Y 125.1045,Z 183,A 69.8747,B 4.4662,C 0.0752,E1 4.5267,E2 382.9596} C_DIS
LIN {X 45.8279,Y 126.4883,Z 183,A 71.1673,B 4.4662,C 0.0774,E1 4.5234,E2 381.7122} C_DIS
LIN {X 42.7638,Y 127.557,Z 183,A 72.5574,B 4.4662,C 0.0759,E1 4.5198,E2 380.3214} C_DIS
LIN {X 40.9809,Y 128.1406,Z 183,A 74.2042,B 4.4664,C 0.0664,E1 4.5151,E2 378.5723} C_DIS
LIN {X 36.0839,Y 129.6049,Z 183,A 75.718,B 4.4664,C 0.0714,E1 4.5113,E2 377.1393} C_DIS
LIN {X 32.6763,Y 130.5064,Z 183,A 77.2062,B 4.4664,C 0.0704,E1 4.5072,E2 375.6531} C_DIS
LIN {X 28.7712,Y 131.4224,Z 183,A 78.9216,B 4.4664,C 0.0691,E1 4.5026,E2 373.9372} C_DIS
LIN {X 25.3924,Y 132.1164,Z 183,A 80.178,B 4.4664,C 0.0704,E1 4.4992,E2 372.7068} C_DIS
LIN {X 22.7164,Y 132.604,Z 183,A 81.5204,B 4.4664,C 0.0679,E1 4.4954,E2 371.3427} C_DIS
LIN {X 19.0371,Y 133.1807,Z 183,A 83.0504,B 4.4664,C 0.0677,E1 4.4912,E2 369.8199} C_DIS
LIN {X 15.9505,Y 133.5856,Z 183,A 84.2452,B 4.4664,C 0.0684,E1 4.488,E2 368.6413} C_DIS
LIN {X 13.2371,Y 133.8823,Z 183,A 85.7749,B 4.4664,C 0.0644,E1 4.4836,E2 367.068} C_DIS
LIN {X 8.1914,Y 134.285,Z 183,A 87.7657,B 4.4664,C 0.0654,E1 4.4781,E2 365.0978} C_DIS
LIN {X 3.8227,Y 134.4803,Z 183,A 89.6093,B 4.4664,C 0.0654,E1 4.473,E2 363.2573} C_DIS
LIN {X 0.0381,Y 134.5365,Z 183,A 91.303,B 4.4664,C 0.0644,E1 4.4682,E2 361.5545} C_DIS
LIN {X -3.9236,Y 134.4775,Z 183,A 92.9387,B 4.4664,C 0.0649,E1 4.4636,E2 359.9256} C_DIS
LIN {X -7.9127,Y 134.3021,Z 183,A 94.6577,B 4.4664,C 0.0649,E1 4.4588,E2 358.2053} C_DIS
LIN {X -12.2943,Y 133.9728,Z 183,A 96.3422,B 4.4664,C 0.0669,E1 4.4542,E2 356.5441} C_DIS
LIN {X -16.7651,Y 133.4877,Z 183,A 98.3772,B 4.4664,C 0.0663,E1 4.4485,E2 354.4958} C_DIS
LIN {X -20.7111,Y 132.9307,Z 183,A 100.1015,B 4.4664,C 0.0666,E1 4.4438,E2 352.769} C_DIS
LIN {X -24.9039,Y 132.2098,Z 183,A 101.7113,B 4.4664,C 0.0692,E1 4.4394,E2 351.1845} C_DIS
LIN {X -28.0903,Y 131.5694,Z 183,A 103.2983,B 4.4664,C 0.0681,E1 4.435,E2 349.574} C_DIS
LIN {X -31.4347,Y 130.8103,Z 183,A 104.7121,B 4.4664,C 0.0694,E1 4.4312,E2 348.1667} C_DIS
LIN {X -33.9693,Y 130.1771,Z 183,A 105.9354,B 4.4664,C 0.0691,E1 4.4278,E2 346.9308} C_DIS
LIN {X -38.1831,Y 129.0026,Z 183,A 108.4026,B 4.4664,C 0.0653,E1 4.421,E2 344.3918} C_DIS
LIN {X -43.0242,Y 127.4702,Z 183,A 110.0739,B 4.4664,C 0.0713,E1 4.4167,E2 342.7812} C_DIS
LIN {X -45.8085,Y 126.4953,Z 183,A 111.803,B 4.4664,C 0.0685,E1 4.4121,E2 340.9959} C_DIS
LIN {X -50.2581,Y 124.794,Z 183,A 113.7185,B 4.4664,C 0.0715,E1 4.4071,E2 339.0955} C_DIS
LIN {X -54.1502,Y 123.1579,Z 183,A 115.2379,B 4.4663,C 0.0757,E1 4.4033,E2 337.6111} C_DIS
LIN {X -57.1723,Y 121.784,Z 183,A 116.6546,B 4.4663,C 0.0773,E1 4.3997,E2 336.195} C_DIS
LIN {X -60.993,Y 119.9136,Z 183,A 118.5319,B 4.4663,C 0.079,E1 4.395,E2 334.311} C_DIS
LIN {X -65.532,Y 117.4975,Z 183,A 120.6785,B 4.4662,C 0.0822,E1 4.3898,E2 332.1713} C_DIS
LIN {X -69.244,Y 115.349,Z 183,A 122.5612,B 4.4662,C 0.0843,E1 4.3852,E2 330.2832} C_DIS
LIN {X -73.0307,Y 112.9891,Z 183,A 124.3637,B 4.4661,C 0.0879,E1 4.381,E2 328.4938} C_DIS
LIN {X -78.04,Y 109.5891,Z 183,A 126.7632,B 4.4659,C 0.0933,E1 4.3756,E2 326.1178} C_DIS
LIN {X -83.165,Y 105.7522,Z 183,A 130.5197,B 4.466,C 0.0901,E1 4.367,E2 322.239} C_DIS
LIN {X -87.477,Y 102.215,Z 183,A 132.3366,B 4.4658,C 0.0985,E1 4.3632,E2 320.4919} C_DIS
LIN {X -93.4975,Y 96.7376,Z 183,A 135.6397,B 4.4657,C 0.1063,E1 4.3565,E2 317.2113} C_DIS
LIN {X -98.2765,Y 91.879,Z 183,A 138.5848,B 4.4655,C 0.1118,E1 4.3508,E2 314.2636} C_DIS
LIN {X -101.0606,Y 88.8075,Z 183,A 140.8201,B 4.4655,C 0.1122,E1 4.3465,E2 311.9729} C_DIS
LIN {X -103.1518,Y 86.3694,Z 183,A 141.9731,B 4.4654,C 0.1166,E1 4.3445,E2 310.8472} C_DIS
LIN {X -107.0026,Y 81.5502,Z 183,A 144.5814,B 4.4652,C 0.1226,E1 4.34,E2 308.2434} C_DIS
LIN {X -109.1073,Y 78.7124,Z 183,A 146.2588,B 4.4652,C 0.1248,E1 4.3372,E2 306.5463} C_DIS
LIN {X -111.3522,Y 75.5026,Z 183,A 148.398,B 4.4652,C 0.1254,E1 4.3337,E2 304.3511} C_DIS
LIN {X -113.7356,Y 71.8622,Z 183,A 149.8243,B 4.4649,C 0.1328,E1 4.3317,E2 302.9783} C_DIS
LIN {X -115.6163,Y 68.7956,Z 183,A 151.4507,B 4.4649,C 0.1358,E1 4.3293,E2 301.3418} C_DIS
LIN {X -117.5361,Y 65.4623,Z 183,A 153.1835,B 4.4647,C 0.1392,E1 4.3269,E2 299.5989} C_DIS
LIN {X -119.7337,Y 61.3462,Z 183,A 155.0932,B 4.4646,C 0.1447,E1 4.3244,E2 297.7001} C_DIS
LIN {X -121.1541,Y 58.4928,Z 183,A 156.3734,B 4.4644,C 0.1487,E1 4.3229,E2 296.4305} C_DIS
LIN {X -122.8037,Y 54.9424,Z 183,A 158.2223,B 4.4644,C 0.1518,E1 4.3207,E2 294.5609} C_DIS
LIN {X -124.1057,Y 51.9346,Z 183,A 159.5286,B 4.4642,C 0.156,E1 4.3193,E2 293.2666} C_DIS
LIN {X -125.0762,Y 49.5582,Z 183,A 160.9494,B 4.4642,C 0.1567,E1 4.3178,E2 291.8069} C_DIS
LIN {X -126.5319,Y 45.707,Z 183,A 162.368,B 4.4639,C 0.1636,E1 4.3164,E2 290.4304} C_DIS
LIN {X -127.2194,Y 43.758,Z 183,A 163.5197,B 4.4639,C 0.1641,E1 4.3154,E2 289.2463} C_DIS
LIN {X -128.5126,Y 39.8016,Z 183,A 165.3669,B 4.4637,C 0.1684,E1 4.3138,E2 287.3914} C_DIS
LIN {X -129.6741,Y 35.8366,Z 183,A 167.2709,B 4.4636,C 0.1723,E1 4.3123,E2 285.4712} C_DIS
LIN {X -130.6961,Y 31.9085,Z 183,A 169.4923,B 4.4636,C 0.1738,E1 4.3108,E2 283.1904} C_DIS
LIN {X -131.7195,Y 27.3824,Z 183,A 171.3962,B 4.4633,C 0.1798,E1 4.3097,E2 281.2971} C_DIS
LIN {X -132.4425,Y 23.6321,Z 183,A 172.5219,B 4.463,C 0.1876,E1 4.3092,E2 280.2343} C_DIS
LIN {X -133.1052,Y 19.5657,Z 183,A 174.5184,B 4.4628,C 0.191,E1 4.3083,E2 278.2095} C_DIS
LIN {X -133.5847,Y 15.9582,Z 183,A 176.0424,B 4.4626,C 0.1955,E1 4.3078,E2 276.6899} C_DIS
LIN {X -133.965,Y 12.3755,Z 183,A 177.6217,B 4.4625,C 0.1995,E1 4.3073,E2 275.1062} C_DIS
LIN {X -134.2666,Y 8.4889,Z 183,A 179.4713,B 4.4623,C 0.203,E1 4.307,E2 273.2344} C_DIS
LIN {X -134.4793,Y 3.86,Z 183,A -178.5887,B 4.462,C 0.2088,E1 4.3068,E2 271.3} C_DIS
LIN {X -134.5378,Y 0.0959,Z 183,A -176.7844,B 4.4619,C 0.2121,E1 4.3068,E2 269.4721} C_DIS
LIN {X -134.4847,Y -3.6668,Z 183,A -175.434,B 4.4616,C 0.2182,E1 4.3068,E2 268.154} C_DIS
LIN {X -134.3675,Y -6.7034,Z 183,A -174.0103,B 4.4615,C 0.221,E1 4.307,E2 266.7151} C_DIS
LIN {X -134.1686,Y -9.9171,Z 183,A -172.4426,B 4.4613,C 0.2236,E1 4.3073,E2 265.1239} C_DIS
LIN {X -133.7868,Y -14.1663,Z 183,A -170.6484,B 4.4611,C 0.2289,E1 4.3078,E2 263.3339} C_DIS
LIN {X -133.4628,Y -16.9554,Z 183,A -169.4802,B 4.4609,C 0.2324,E1 4.3082,E2 262.1699} C_DIS
LIN {X -133.0691,Y -19.817,Z 183,A -167.9733,B 4.4608,C 0.2341,E1 4.3088,E2 260.6293} C_DIS
LIN {X -132.4149,Y -23.7868,Z 183,A -166.3631,B 4.4605,C 0.2395,E1 4.3095,E2 259.033} C_DIS
LIN {X -131.7237,Y -27.3613,Z 183,A -164.6374,B 4.4603,C 0.2426,E1 4.3105,E2 257.2864} C_DIS
LIN {X -130.8224,Y -31.3847,Z 183,A -163.0822,B 4.46,C 0.2488,E1 4.3115,E2 255.7573} C_DIS
LIN {X -129.6801,Y -35.815,Z 183,A -161.0518,B 4.4597,C 0.2536,E1 4.3129,E2 253.7179} C_DIS
LIN {X -128.7657,Y -38.9745,Z 183,A -159.5992,B 4.4595,C 0.257,E1 4.3141,E2 252.2597} C_DIS
LIN {X -127.7279,Y -42.2505,Z 183,A -158.0203,B 4.4593,C 0.2601,E1 4.3154,E2 250.6671} C_DIS
LIN {X -125.5559,Y -48.3255,Z 183,A -155.0535,B 4.459,C 0.2659,E1 4.3183,E2 247.6743} C_DIS
LIN {X -124.2333,Y -51.6291,Z 183,A -153.5963,B 4.4587,C 0.2702,E1 4.3198,E2 246.2252} C_DIS
LIN {X -123.1412,Y -54.1878,Z 183,A -152.2372,B 4.4587,C 0.2721,E1 4.3214,E2 244.8448} C_DIS
LIN {X -121.439,Y -57.8964,Z 183,A -150.6295,B 4.4583,C 0.2774,E1 4.3233,E2 243.2542} C_DIS
LIN {X -120.0334,Y -60.7575,Z 183,A -149.0171,B 4.4583,C 0.279,E1 4.3253,E2 241.6103} C_DIS
LIN {X -117.7055,Y -65.1566,Z 183,A -147.1943,B 4.4577,C 0.2863,E1 4.3277,E2 239.8258} C_DIS
LIN {X -115.9837,Y -68.1743,Z 183,A -145.5292,B 4.4577,C 0.2885,E1 4.33,E2 238.1381} C_DIS
LIN {X -114.0449,Y -71.3712,Z 183,A -143.856,B 4.4574,C 0.2917,E1 4.3325,E2 236.4552} C_DIS
LIN {X -112.2322,Y -74.1886,Z 183,A -142.556,B 4.4571,C 0.296,E1 4.3345,E2 235.1718} C_DIS
LIN {X -110.5773,Y -76.6333,Z 183,A -141.1462,B 4.4571,C 0.2977,E1 4.3367,E2 233.7432} C_DIS
LIN {X -108.4902,Y -79.5603,Z 183,A -139.5754,B 4.4568,C 0.3009,E1 4.3393,E2 232.1677} C_DIS
LIN {X -106.2047,Y -82.5867,Z 183,A -137.8379,B 4.4566,C 0.3035,E1 4.3423,E2 230.4152} C_DIS
LIN {X -103.6647,Y -85.753,Z 183,A -136.0444,B 4.4564,C 0.3067,E1 4.3454,E2 228.614} C_DIS
LIN {X -100.922,Y -88.9648,Z 183,A -134.1154,B 4.4562,C 0.3094,E1 4.349,E2 226.6689} C_DIS
LIN {X -97.6942,Y -92.4979,Z 183,A -132.1412,B 4.4559,C 0.314,E1 4.3527,E2 224.7032} C_DIS
LIN {X -95.0114,Y -95.2516,Z 183,A -130.372,B 4.4557,C 0.3162,E1 4.3562,E2 222.9176} C_DIS
LIN {X -91.7143,Y -98.4299,Z 183,A -128.3971,B 4.4555,C 0.3196,E1 4.3603,E2 220.9399} C_DIS
LIN {X -88.5066,Y -101.3239,Z 183,A -126.5556,B 4.4552,C 0.3229,E1 4.3641,E2 219.0985} C_DIS
LIN {X -85.4012,Y -103.9553,Z 183,A -124.7146,B 4.4551,C 0.3251,E1 4.3681,E2 217.2439} C_DIS
LIN {X -81.772,Y -106.833,Z 183,A -122.7463,B 4.4549,C 0.3283,E1 4.3724,E2 215.2763} C_DIS
LIN {X -78.0767,Y -109.5629,Z 183,A -120.7589,B 4.4546,C 0.3312,E1 4.3769,E2 213.285} C_DIS
LIN {X -74.4536,Y -112.0567,Z 183,A -118.9478,B 4.4544,C 0.3345,E1 4.3811,E2 211.4819} C_DIS
LIN {X -71.8823,Y -113.7229,Z 183,A -117.7329,B 4.4542,C 0.3371,E1 4.3839,E2 210.2785} C_DIS
LIN {X -69.1417,Y -115.41,Z 183,A -116.2538,B 4.4542,C 0.338,E1 4.3875,E2 208.7855} C_DIS
LIN {X -65.1653,Y -117.7007,Z 183,A -114.2463,B 4.454,C 0.3401,E1 4.3924,E2 206.7712} C_DIS
LIN {X -61.5061,Y -119.6523,Z 183,A -112.3392,B 4.454,C 0.341,E1 4.3971,E2 204.8458} C_DIS
LIN {X -58.3956,Y -121.2005,Z 183,A -110.897,B 4.4538,C 0.343,E1 4.4008,E2 203.4083} C_DIS
LIN {X -54.8804,Y -122.8314,Z 183,A -109.2226,B 4.4536,C 0.3445,E1 4.405,E2 201.7306} C_DIS
LIN {X -50.9319,Y -124.5224,Z 183,A -107.2652,B 4.4536,C 0.3452,E1 4.4101,E2 199.7565} C_DIS
LIN {X -47.7719,Y -125.7683,Z 183,A -105.8423,B 4.4535,C 0.3467,E1 4.4138,E2 198.3364} C_DIS
LIN {X -44.0107,Y -127.1318,Z 183,A -103.5797,B 4.4538,C 0.343,E1 4.42,E2 196.0012} C_DIS
LIN {X -39.0431,Y -128.7448,Z 183,A -101.9995,B 4.4532,C 0.3505,E1 4.424,E2 194.5038} C_DIS
LIN {X -35.62,Y -129.7347,Z 183,A -100.3292,B 4.4532,C 0.35,E1 4.4285,E2 192.8135} C_DIS
LIN {X -31.6366,Y -130.7617,Z 183,A -98.6809,B 4.4531,C 0.352,E1 4.433,E2 191.178} C_DIS
LIN {X -28.2492,Y -131.5351,Z 183,A -97.1878,B 4.4531,C 0.3526,E1 4.437,E2 189.6828} C_DIS
LIN {X -24.0631,Y -132.3654,Z 183,A -95.3837,B 4.4529,C 0.3534,E1 4.442,E2 187.8798} C_DIS
LIN {X -20.6161,Y -132.9454,Z 183,A -93.8846,B 4.4529,C 0.3538,E1 4.4461,E2 186.3789} C_DIS
LIN {X -16.9595,Y -133.4623,Z 183,A -92.0617,B 4.4531,C 0.3517,E1 4.4513,E2 184.5231} C_DIS
LIN {X -11.4589,Y -134.0457,Z 183,A -90.0816,B 4.4528,C 0.3558,E1 4.4566,E2 182.5906} C_DIS
LIN {X -8.1729,Y -134.2861,Z 183,A -88.5488,B 4.4528,C 0.3545,E1 4.461,E2 181.0405} C_DIS
LIN {X -4.231,Y -134.469,Z 183,A -86.7276,B 4.453,C 0.3531,E1 4.4661,E2 179.2004} C_DIS
LIN {X 0.9664,Y -134.5293,Z 183,A -85.4345,B 4.4522,C 0.3621,E1 4.4694,E2 178.0243} C_DIS
Enddeposition()
LIN {X 0.9664,Y -134.5293,Z 183,A -85.4346,B 4.4522,C 0.3621,E1 4.4694,E2 178.0245} C_DIS
Startdeposition()
$VEL.CP = VEL_PRINT
LIN {X -3.6096,Y -135.3876,Z 183,A -87.2636,B 4.4522,C 0.3637,E1 4.4643,E2 179.8728} C_DIS
LIN {X -8.1307,Y -135.1914,Z 183,A -88.8921,B 4.4524,C 0.3609,E1 4.4599,E2 181.4653} C_DIS
LIN {X -11.1082,Y -134.9796,Z 183,A -90.4513,B 4.4522,C 0.3637,E1 4.4554,E2 183.0633} C_DIS
LIN {X -19.0968,Y -134.0824,Z 183,A -93.509,B 4.4525,C 0.3597,E1 4.4471,E2 186.0782} C_DIS
LIN {X -22.1706,Y -133.6085,Z 183,A -95.133,B 4.4523,C 0.3623,E1 4.4425,E2 187.7424} C_DIS
LIN {X -26.0113,Y -132.9154,Z 183,A -96.7493,B 4.4523,C 0.3613,E1 4.438,E2 189.3548} C_DIS
LIN {X -29.3678,Y -132.2154,Z 183,A -98.4161,B 4.4523,C 0.3627,E1 4.4334,E2 191.0498} C_DIS
LIN {X -33.5344,Y -131.2182,Z 183,A -100.0603,B 4.4525,C 0.3601,E1 4.429,E2 192.673} C_DIS
LIN {X -36.9555,Y -130.2968,Z 183,A -101.6961,B 4.4525,C 0.3604,E1 4.4245,E2 194.3266} C_DIS
LIN {X -41.5266,Y -128.9122,Z 183,A -103.8055,B 4.4525,C 0.3598,E1 4.4189,E2 196.4479} C_DIS
LIN {X -46.2153,Y -127.3064,Z 183,A -105.7382,B 4.4528,C 0.3566,E1 4.4138,E2 198.36} C_DIS
LIN {X -49.7411,Y -125.9723,Z 183,A -107.3188,B 4.4528,C 0.355,E1 4.4097,E2 199.9392} C_DIS
LIN {X -52.7114,Y -124.7578,Z 183,A -108.6789,B 4.453,C 0.3537,E1 4.4062,E2 201.2998} C_DIS
LIN {X -55.605,Y -123.4944,Z 183,A -110.0349,B 4.453,C 0.3525,E1 4.4027,E2 202.6586} C_DIS
LIN {X -58.4596,Y -122.1685,Z 183,A -111.4693,B 4.4531,C 0.352,E1 4.3991,E2 204.1061} C_DIS
LIN {X -62.3692,Y -120.2214,Z 183,A -113.3839,B 4.4533,C 0.3504,E1 4.3943,E2 206.0295} C_DIS
LIN {X -66.2006,Y -118.1555,Z 183,A -115.3231,B 4.4533,C 0.3489,E1 4.3895,E2 207.9814} C_DIS
LIN {X -70.0843,Y -115.8939,Z 183,A -117.1944,B 4.4536,C 0.3461,E1 4.385,E2 209.8489} C_DIS
LIN {X -73.2499,Y -113.9199,Z 183,A -118.785,B 4.4538,C 0.344,E1 4.3813,E2 211.4411} C_DIS
LIN {X -76.9697,Y -111.4407,Z 183,A -120.7017,B 4.454,C 0.3414,E1 4.3768,E2 213.361} C_DIS
LIN {X -80.3779,Y -109.0076,Z 183,A -122.4994,B 4.4542,C 0.3388,E1 4.3728,E2 215.1619} C_DIS
LIN {X -83.7114,Y -106.4688,Z 183,A -124.3186,B 4.4543,C 0.3363,E1 4.3687,E2 216.9869} C_DIS
LIN {X -87.2333,Y -103.6031,Z 183,A -126.285,B 4.4546,C 0.3333,E1 4.3645,E2 218.9589} C_DIS
LIN {X -90.677,Y -100.6035,Z 183,A -128.2696,B 4.4548,C 0.3303,E1 4.3603,E2 220.9499} C_DIS
LIN {X -94.3177,Y -97.1977,Z 183,A -130.4007,B 4.4551,C 0.3265,E1 4.356,E2 223.0834} C_DIS
LIN {X -97.4002,Y -94.1086,Z 183,A -132.2655,B 4.4553,C 0.3231,E1 4.3523,E2 224.9502} C_DIS
LIN {X -101.4347,Y -89.7453,Z 183,A -134.6486,B 4.4558,C 0.317,E1 4.3479,E2 227.3162} C_DIS
LIN {X -103.5279,Y -87.323,Z 183,A -136.2263,B 4.4558,C 0.3159,E1 4.345,E2 228.9218} C_DIS
LIN {X -106.2337,Y -84.0107,Z 183,A -138.1341,B 4.4561,C 0.3127,E1 4.3416,E2 230.8416} C_DIS
LIN {X -108.9226,Y -80.4935,Z 183,A -140.0857,B 4.4563,C 0.3091,E1 4.3383,E2 232.8025} C_DIS
LIN {X -111.9985,Y -76.1552,Z 183,A -142.3438,B 4.4567,C 0.3041,E1 4.3347,E2 235.061} C_DIS
LIN {X -114.384,Y -72.523,Z 183,A -144.2551,B 4.4569,C 0.3003,E1 4.3318,E2 236.9807} C_DIS
LIN {X -116.7627,Y -68.6271,Z 183,A -146.6164,B 4.457,C 0.2988,E1 4.3284,E2 239.3951} C_DIS
LIN {X -118.8615,Y -64.9242,Z 183,A -147.6738,B 4.4576,C 0.2892,E1 4.3271,E2 240.3586} C_DIS
LIN {X -120.8839,Y -61.073,Z 183,A -149.9527,B 4.4577,C 0.2877,E1 4.3241,E2 242.6919} C_DIS
LIN {X -122.8627,Y -56.9862,Z 183,A -151.8952,B 4.458,C 0.283,E1 4.3217,E2 244.6363} C_DIS
LIN {X -124.4371,Y -53.4619,Z 183,A -153.5348,B 4.4583,C 0.2788,E1 4.3199,E2 246.2759} C_DIS
LIN {X -125.7022,Y -50.4153,Z 183,A -154.9708,B 4.4585,C 0.2755,E1 4.3183,E2 247.7163} C_DIS
LIN {X -127.1094,Y -46.7603,Z 183,A -157.6719,B 4.4583,C 0.2782,E1 4.3157,E2 250.5461} C_DIS
LIN {X -129.2948,Y -40.3237,Z 183,A -159.6417,B 4.4592,C 0.2644,E1 4.314,E2 252.4023} C_DIS
LIN {X -129.9747,Y -38.0695,Z 183,A -161.399,B 4.459,C 0.2668,E1 4.3126,E2 254.2533} C_DIS
LIN {X -131.4166,Y -32.7526,Z 183,A -162.993,B 4.4597,C 0.2556,E1 4.3116,E2 255.7548} C_DIS
LIN {X -132.0265,Y -30.1948,Z 183,A -164.2122,B 4.4598,C 0.2532,E1 4.3108,E2 256.9866} C_DIS
LIN {X -132.7292,Y -26.9388,Z 183,A -165.6677,B 4.46,C 0.2496,E1 4.3099,E2 258.4471} C_DIS
LIN {X -133.3593,Y -23.6241,Z 183,A -167.119,B 4.4602,C 0.2458,E1 4.3092,E2 259.9004} C_DIS
LIN {X -133.9088,Y -20.2825,Z 183,A -168.7455,B 4.4604,C 0.2431,E1 4.3085,E2 261.55} C_DIS
LIN {X -134.4722,Y -16.1247,Z 183,A -170.474,B 4.4607,C 0.2378,E1 4.3079,E2 263.2716} C_DIS
LIN {X -134.8425,Y -12.6636,Z 183,A -171.9991,B 4.4609,C 0.234,E1 4.3074,E2 264.8022} C_DIS
LIN {X -135.1636,Y -8.5825,Z 183,A -173.8112,B 4.4611,C 0.2296,E1 4.3071,E2 266.623} C_DIS
LIN {X -135.3569,Y -4.6575,Z 183,A -175.6246,B 4.4613,C 0.2259,E1 4.3069,E2 268.454} C_DIS
LIN {X -135.4361,Y -0.5154,Z 183,A -177.3057,B 4.4616,C 0.2205,E1 4.3069,E2 270.125} C_DIS
LIN {X -135.3928,Y 3.4223,Z 183,A -179.0779,B 4.4618,C 0.2164,E1 4.3069,E2 271.9091} C_DIS
LIN {X -135.2479,Y 7.1354,Z 183,A 179.3151,B 4.462,C 0.2122,E1 4.3071,E2 273.5192} C_DIS
LIN {X -134.9548,Y 11.4008,Z 183,A 177.4608,B 4.4622,C 0.2074,E1 4.3075,E2 275.3778} C_DIS
LIN {X -134.6547,Y 14.5225,Z 183,A 176.0831,B 4.4623,C 0.204,E1 4.3079,E2 276.7608} C_DIS
LIN {X -134.1641,Y 18.5251,Z 183,A 174.2217,B 4.4625,C 0.2002,E1 4.3086,E2 278.6399} C_DIS
LIN {X -133.5682,Y 22.4123,Z 183,A 172.6129,B 4.4627,C 0.1952,E1 4.3093,E2 280.2407} C_DIS
LIN {X -132.8858,Y 26.1658,Z 183,A 170.978,B 4.4629,C 0.1908,E1 4.3101,E2 281.877} C_DIS
LIN {X -131.5677,Y 32.1376,Z 183,A 168.2989,B 4.4632,C 0.1842,E1 4.3118,E2 284.5652} C_DIS
LIN {X -130.6176,Y 35.8082,Z 183,A 166.0931,B 4.4632,C 0.1837,E1 4.3134,E2 286.843} C_DIS
LIN {X -129.4017,Y 39.9755,Z 183,A 164.7475,B 4.4636,C 0.1756,E1 4.3145,E2 288.1275} C_DIS
LIN {X -127.6454,Y 45.2743,Z 183,A 162.3588,B 4.4638,C 0.1694,E1 4.3166,E2 290.5176} C_DIS
LIN {X -126.7461,Y 47.7302,Z 183,A 161.1287,B 4.4638,C 0.1673,E1 4.3178,E2 291.7618} C_DIS
LIN {X -125.6537,Y 50.5355,Z 183,A 159.8464,B 4.464,C 0.164,E1 4.3191,E2 293.0441} C_DIS
LIN {X -124.384,Y 53.5846,Z 183,A 157.8466,B 4.464,C 0.1643,E1 4.3214,E2 295.1156} C_DIS
LIN {X -122.4897,Y 57.7872,Z 183,A 156.462,B 4.4643,C 0.1556,E1 4.323,E2 296.4303} C_DIS
LIN {X -121.3299,Y 60.1813,Z 183,A 155.2027,B 4.4643,C 0.1536,E1 4.3245,E2 297.7049} C_DIS
LIN {X -119.678,Y 63.404,Z 183,A 153.6564,B 4.4645,C 0.1498,E1 4.3265,E2 299.2517} C_DIS
LIN {X -117.7373,Y 66.9416,Z 183,A 151.8052,B 4.4645,C 0.1466,E1 4.3291,E2 301.119} C_DIS
LIN {X -115.5557,Y 70.6408,Z 183,A 149.9542,B 4.4647,C 0.1424,E1 4.3317,E2 302.9726} C_DIS
LIN {X -113.0509,Y 74.5835,Z 183,A 147.2427,B 4.4647,C 0.1428,E1 4.336,E2 305.7706} C_DIS
LIN {X -109.8817,Y 79.1792,Z 183,A 145.7533,B 4.4651,C 0.1314,E1 4.3382,E2 307.1534} C_DIS
LIN {X -108.162,Y 81.5119,Z 183,A 143.9296,B 4.4651,C 0.1327,E1 4.3414,E2 309.048} C_DIS
LIN {X -105.9248,Y 84.3987,Z 183,A 142.5261,B 4.4651,C 0.1283,E1 4.3438,E2 310.4334} C_DIS
LIN {X -103.6073,Y 87.2283,Z 183,A 140.3974,B 4.4651,C 0.1291,E1 4.3478,E2 312.6302} C_DIS
LIN {X -99.9624,Y 91.383,Z 183,A 138.7504,B 4.4654,C 0.1193,E1 4.3507,E2 314.1929} C_DIS
LIN {X -97.2851,Y 94.2275,Z 183,A 136.8702,B 4.4654,C 0.1176,E1 4.3544,E2 316.099} C_DIS
LIN {X -93.5774,Y 97.9105,Z 183,A 134.2981,B 4.4654,C 0.1159,E1 4.3596,E2 318.7124} C_DIS
LIN {X -90.4725,Y 100.7866,Z 183,A 133.1131,B 4.4657,C 0.1082,E1 4.3619,E2 319.8236} C_DIS
LIN {X -88.0771,Y 102.8873,Z 183,A 131.4846,B 4.4657,C 0.1078,E1 4.3654,E2 321.4848} C_DIS
LIN {X -83.2002,Y 106.8691,Z 183,A 128.2396,B 4.4657,C 0.1075,E1 4.3727,E2 324.7969} C_DIS
LIN {X -79.2583,Y 109.8244,Z 183,A 126.8321,B 4.4659,C 0.099,E1 4.3756,E2 326.1222} C_DIS
LIN {X -76.3124,Y 111.8918,Z 183,A 124.8827,B 4.4659,C 0.0998,E1 4.3802,E2 328.1215} C_DIS
LIN {X -73.6131,Y 113.6853,Z 183,A 123.8561,B 4.4659,C 0.0951,E1 4.3825,E2 329.1059} C_DIS
LIN {X -70.5128,Y 115.6342,Z 183,A 122.1479,B 4.466,C 0.0941,E1 4.3866,E2 330.8321} C_DIS
LIN {X -66.9969,Y 117.7057,Z 183,A 120.376,B 4.466,C 0.0921,E1 4.3909,E2 332.6081} C_DIS
LIN {X -60.9812,Y 120.9306,Z 183,A 117.545,B 4.4661,C 0.088,E1 4.3979,E2 335.4302} C_DIS
LIN {X -58.2194,Y 122.2833,Z 183,A 116.1777,B 4.4661,C 0.087,E1 4.4014,E2 336.8046} C_DIS
LIN {X -54.6737,Y 123.9109,Z 183,A 114.3656,B 4.4661,C 0.0864,E1 4.406,E2 338.6349} C_DIS
LIN {X -50.2112,Y 125.7833,Z 183,A 111.857,B 4.4661,C 0.0881,E1 4.4127,E2 341.1967} C_DIS
LIN {X -45.5904,Y 127.5317,Z 183,A 110.3769,B 4.4663,C 0.0812,E1 4.4164,E2 342.6031} C_DIS
LIN {X -42.6567,Y 128.5423,Z 183,A 108.7725,B 4.4663,C 0.0825,E1 4.4207,E2 344.2415} C_DIS
LIN {X -37.5825,Y 130.1173,Z 183,A 106.8009,B 4.4663,C 0.0785,E1 4.4259,E2 346.1788} C_DIS
LIN {X -34.6475,Y 130.9287,Z 183,A 105.4425,B 4.4663,C 0.0782,E1 4.4296,E2 347.5448} C_DIS
LIN {X -31.2095,Y 131.7915,Z 183,A 103.814,B 4.4663,C 0.0784,E1 4.434,E2 349.1878} C_DIS
LIN {X -26.9271,Y 132.7316,Z 183,A 102.109,B 4.4663,C 0.0761,E1 4.4386,E2 350.8739} C_DIS
LIN {X -23.611,Y 133.3617,Z 183,A 100.5979,B 4.4663,C 0.0762,E1 4.4428,E2 352.3941} C_DIS
LIN {X -19.2835,Y 134.0557,Z 183,A 98.7778,B 4.4663,C 0.0752,E1 4.4478,E2 354.2091} C_DIS
LIN {X -15.8248,Y 134.508,Z 183,A 96.849,B 4.4663,C 0.0789,E1 4.4533,E2 356.191} C_DIS
LIN {X -11.6998,Y 134.9296,Z 183,A 95.4943,B 4.4663,C 0.075,E1 4.457,E2 357.4974} C_DIS
LIN {X -8.2666,Y 135.1831,Z 183,A 94.0927,B 4.4663,C 0.0743,E1 4.4608,E2 358.8918} C_DIS
LIN {X -4.2078,Y 135.371,Z 183,A 91.9952,B 4.4663,C 0.0777,E1 4.4668,E2 361.0336} C_DIS
LIN {X -0.547,Y 135.4347,Z 183,A 90.541,B 4.4663,C 0.0769,E1 4.4709,E2 362.4759} C_DIS
LIN {X 2.7066,Y 135.4094,Z 183,A 89.511,B 4.4663,C 0.0738,E1 4.4736,E2 363.4641} C_DIS
LIN {X 5.4883,Y 135.3245,Z 183,A 88.2108,B 4.4663,C 0.0752,E1 4.4773,E2 364.7783} C_DIS
LIN {X 9.9562,Y 135.0692,Z 183,A 85.7268,B 4.4663,C 0.0813,E1 4.4844,E2 367.3318} C_DIS
LIN {X 15.2443,Y 134.577,Z 183,A 84.1771,B 4.4663,C 0.0754,E1 4.4885,E2 368.798} C_DIS
LIN {X 18.5064,Y 134.1667,Z 183,A 82.6587,B 4.4663,C 0.0772,E1 4.4927,E2 370.3311} C_DIS
LIN {X 22.6336,Y 133.5313,Z 183,A 80.9183,B 4.4663,C 0.0779,E1 4.4975,E2 372.0677} C_DIS
LIN {X 26.7448,Y 132.7687,Z 183,A 79.203,B 4.4663,C 0.0784,E1 4.5022,E2 373.7761} C_DIS
LIN {X 30.6668,Y 131.9187,Z 183,A 77.6087,B 4.4663,C 0.0785,E1 4.5065,E2 375.3577} C_DIS
LIN {X 33.5705,Y 131.209,Z 183,A 76.3191,B 4.4663,C 0.0797,E1 4.51,E2 376.6499} C_DIS
LIN {X 36.8222,Y 130.3341,Z 183,A 74.8933,B 4.4663,C 0.0809,E1 4.5139,E2 378.0756} C_DIS
LIN {X 41.3918,Y 128.9552,Z 183,A 72.8923,B 4.4663,C 0.0825,E1 4.5192,E2 380.0739} C_DIS
LIN {X 45.0895,Y 127.7115,Z 183,A 71.0884,B 4.4662,C 0.0857,E1 4.524,E2 381.896} C_DIS
LIN {X 49.1157,Y 126.2154,Z 183,A 69.4877,B 4.4662,C 0.0854,E1 4.5281,E2 383.4704} C_DIS
LIN {X 52.0464,Y 125.0355,Z 183,A 68.166,B 4.4662,C 0.0867,E1 4.5315,E2 384.7901} C_DIS
LIN {X 55.148,Y 123.6988,Z 183,A 66.6991,B 4.4662,C 0.0888,E1 4.5353,E2 386.2614} C_DIS
LIN {X 58.5049,Y 122.1468,Z 183,A 65.2106,B 4.4661,C 0.09,E1 4.539,E2 387.7407} C_DIS
LIN {X 61.4966,Y 120.6683,Z 183,A 63.7729,B 4.4661,C 0.0921,E1 4.5426,E2 389.1813} C_DIS
LIN {X 65.0351,Y 118.8011,Z 183,A 62.1086,B 4.4661,C 0.0942,E1 4.5467,E2 390.8423} C_DIS
LIN {X 68.2553,Y 116.9811,Z 183,A 60.4769,B 4.4659,C 0.0972,E1 4.5507,E2 392.482} C_DIS
LIN {X 72.0937,Y 114.6549,Z 183,A 58.6406,B 4.4659,C 0.0994,E1 4.555,E2 394.3107} C_DIS
LIN {X 75.7405,Y 112.2793,Z 183,A 56.8368,B 4.4659,C 0.102,E1 4.5592,E2 396.11} C_DIS
LIN {X 79.329,Y 109.7732,Z 183,A 55.0295,B 4.4658,C 0.1046,E1 4.5633,E2 397.912} C_DIS
LIN {X 83.0168,Y 107.0113,Z 183,A 53.1947,B 4.4658,C 0.1067,E1 4.5674,E2 399.7332} C_DIS
LIN {X 86.4324,Y 104.272,Z 183,A 51.3064,B 4.4656,C 0.1105,E1 4.5715,E2 401.626} C_DIS
LIN {X 89.8614,Y 101.332,Z 183,A 48.7799,B 4.4654,C 0.1212,E1 4.5769,E2 404.2268} C_DIS
LIN {X 94.0589,Y 97.4483,Z 183,A 47.0584,B 4.4654,C 0.1179,E1 4.5803,E2 405.8648} C_DIS
LIN {X 98.6415,Y 92.8067,Z 183,A 44.4174,B 4.4654,C 0.1222,E1 4.5854,E2 408.4921} C_DIS
LIN {X 101.5718,Y 89.5902,Z 183,A 42.5811,B 4.4652,C 0.1261,E1 4.5888,E2 410.3283} C_DIS
LIN {X 105.2023,Y 85.2984,Z 183,A 40.5242,B 4.4652,C 0.1275,E1 4.5924,E2 412.3467} C_DIS
LIN {X 107.4884,Y 82.3982,Z 183,A 38.8863,B 4.4651,C 0.1319,E1 4.5953,E2 413.9943} C_DIS
LIN {X 109.5097,Y 79.6925,Z 183,A 37.3052,B 4.4649,C 0.137,E1 4.5979,E2 415.5944} C_DIS
LIN {X 112.147,Y 75.9359,Z 183,A 35.5498,B 4.4649,C 0.1393,E1 4.6007,E2 417.3277} C_DIS
LIN {X 114.0751,Y 73.0074,Z 183,A 34.0537,B 4.4647,C 0.143,E1 4.6029,E2 418.8258} C_DIS
LIN {X 116.2565,Y 69.4813,Z 183,A 32.0888,B 4.4645,C 0.1499,E1 4.6058,E2 420.8172} C_DIS
LIN {X 117.929,Y 66.6036,Z 183,A 31.2223,B 4.4645,C 0.1467,E1 4.6069,E2 421.618} C_DIS
LIN {X 120.0487,Y 62.698,Z 183,A 29.1677,B 4.4644,C 0.1536,E1 4.6097,E2 423.6948} C_DIS
LIN {X 121.9546,Y 58.9074,Z 183,A 27.2196,B 4.4641,C 0.16,E1 4.6121,E2 425.6624} C_DIS
LIN {X 123.8168,Y 54.8842,Z 183,A 25.6223,B 4.4641,C 0.1614,E1 4.6139,E2 427.2265} C_DIS
LIN {X 125.15,Y 51.7722,Z 183,A 24.0933,B 4.4639,C 0.1664,E1 4.6156,E2 428.7681} C_DIS
LIN {X 126.7767,Y 47.6485,Z 183,A 21.9825,B 4.4636,C 0.1743,E1 4.6177,E2 430.9086} C_DIS
LIN {X 128.1738,Y 43.7559,Z 183,A 20.7185,B 4.4636,C 0.1729,E1 4.6188,E2 432.114} C_DIS
LIN {X 129.1874,Y 40.665,Z 183,A 19.2804,B 4.4635,C 0.1774,E1 4.62,E2 433.5605} C_DIS
LIN {X 130.3823,Y 36.6498,Z 183,A 17.6369,B 4.4634,C 0.1806,E1 4.6213,E2 435.1891} C_DIS
LIN {X 131.2631,Y 33.3576,Z 183,A 16.2059,B 4.4632,C 0.1844,E1 4.6223,E2 436.6196} C_DIS
LIN {X 132.2948,Y 29.0001,Z 183,A 14.3553,B 4.463,C 0.1891,E1 4.6235,E2 438.4659} C_DIS
LIN {X 133.0462,Y 25.327,Z 183,A 12.9163,B 4.4629,C 0.1917,E1 4.6242,E2 439.8876} C_DIS
LIN {X 133.6086,Y 22.1697,Z 183,A 11.6185,B 4.4628,C 0.1947,E1 4.6248,E2 441.179} C_DIS
LIN {X 134.0894,Y 19.0474,Z 183,A 10.2415,B 4.4626,C 0.199,E1 4.6254,E2 442.5619} C_DIS
LIN {X 134.7364,Y 13.763,Z 183,A 8.1191,B 4.4624,C 0.2037,E1 4.6261,E2 444.6696} C_DIS
LIN {X 135.2374,Y 7.3444,Z 183,A 5.5653,B 4.4621,C 0.2092,E1 4.6266,E2 447.2042} C_DIS
LIN {X 135.3737,Y 4.1104,Z 183,A 3.5896,B 4.4615,C 0.2208,E1 4.6268,E2 449.2561} C_DIS
LIN {X 135.4355,Y -0.5929,Z 183,A 1.998,B 4.4615,C 0.2214,E1 4.6268,E2 450.7998} C_DIS
LIN {X 135.3611,Y -4.5508,Z 183,A 0.47,B 4.4614,C 0.2243,E1 4.6267,E2 452.3108} C_DIS
LIN {X 135.1602,Y -8.6384,Z 183,A -1.1614,B 4.4612,C 0.2279,E1 4.6264,E2 453.931} C_DIS
LIN {X 134.3963,Y -16.7611,Z 183,A -4.4033,B 4.4608,C 0.235,E1 4.6255,E2 457.1493} C_DIS
LIN {X 133.7908,Y -21.045,Z 183,A -6.3056,B 4.4605,C 0.241,E1 4.6247,E2 459.062} C_DIS
LIN {X 133.0307,Y -25.4082,Z 183,A -8.035,B 4.4603,C 0.2444,E1 4.6239,E2 460.7748} C_DIS
LIN {X 132.2907,Y -29.0193,Z 183,A -9.5602,B 4.4601,C 0.2483,E1 4.623,E2 462.297} C_DIS
LIN {X 131.3133,Y -33.1597,Z 183,A -11.2937,B 4.4599,C 0.2525,E1 4.6219,E2 464.0236} C_DIS
LIN {X 130.3947,Y -36.6055,Z 183,A -12.7592,B 4.4597,C 0.2561,E1 4.6208,E2 465.4849} C_DIS
LIN {X 129.5031,Y -39.6441,Z 183,A -14.0557,B 4.4595,C 0.2592,E1 4.6198,E2 466.777} C_DIS
LIN {X 128.059,Y -44.0871,Z 183,A -16.2541,B 4.459,C 0.2674,E1 4.6178,E2 469.0051} C_DIS
LIN {X 126.9536,Y -47.1762,Z 183,A -17.1342,B 4.4592,C 0.2646,E1 4.617,E2 469.8222} C_DIS
LIN {X 125.9773,Y -49.7283,Z 183,A -18.6634,B 4.4587,C 0.2725,E1 4.6154,E2 471.3996} C_DIS
LIN {X 124.2774,Y -53.8313,Z 183,A -20.2834,B 4.4586,C 0.2741,E1 4.6137,E2 472.9885} C_DIS
LIN {X 122.8408,Y -57.0337,Z 183,A -21.7154,B 4.4584,C 0.2774,E1 4.612,E2 474.4151} C_DIS
LIN {X 121.3374,Y -60.1661,Z 183,A -23.1695,B 4.4582,C 0.2809,E1 4.6102,E2 475.8684} C_DIS
LIN {X 119.151,Y -64.392,Z 183,A -25.5324,B 4.4576,C 0.2905,E1 4.6071,E2 478.2773} C_DIS
LIN {X 117.1319,Y -67.9952,Z 183,A -26.8673,B 4.4576,C 0.2897,E1 4.6053,E2 479.5616} C_DIS
LIN {X 114.8316,Y -71.8122,Z 183,A -28.6777,B 4.4574,C 0.2934,E1 4.6027,E2 481.3641} C_DIS
LIN {X 112.2781,Y -75.7422,Z 183,A -30.8401,B 4.4569,C 0.3004,E1 4.5993,E2 483.551} C_DIS
LIN {X 110.3958,Y -78.4606,Z 183,A -32.0277,B 4.4569,C 0.3011,E1 4.5974,E2 484.713} C_DIS
LIN {X 108.1888,Y -81.4765,Z 183,A -33.5482,B 4.4567,C 0.304,E1 4.5949,E2 486.2272} C_DIS
LIN {X 105.5405,Y -84.8789,Z 183,A -35.3008,B 4.4564,C 0.3073,E1 4.5919,E2 487.9723} C_DIS
LIN {X 102.7859,Y -88.1948,Z 183,A -37.1241,B 4.4562,C 0.3114,E1 4.5886,E2 489.7971} C_DIS
LIN {X 99.7007,Y -91.6677,Z 183,A -38.996,B 4.4559,C 0.3145,E1 4.5851,E2 491.6588} C_DIS
LIN {X 96.7996,Y -94.7263,Z 183,A -40.7683,B 4.4557,C 0.3181,E1 4.5817,E2 493.4312} C_DIS
LIN {X 93.5277,Y -97.9581,Z 183,A -42.6559,B 4.4554,C 0.3214,E1 4.5779,E2 495.313} C_DIS
LIN {X 90.1135,Y -101.1082,Z 183,A -44.5818,B 4.4552,C 0.3248,E1 4.5739,E2 497.2355} C_DIS
LIN {X 86.7267,Y -104.0281,Z 183,A -46.4456,B 4.455,C 0.3281,E1 4.5699,E2 499.0974} C_DIS
LIN {X 83.3075,Y -106.786,Z 183,A -48.2696,B 4.4547,C 0.3312,E1 4.566,E2 500.9184} C_DIS
LIN {X 79.7789,Y -109.4471,Z 183,A -50.0824,B 4.4545,C 0.3338,E1 4.5619,E2 502.7255} C_DIS
LIN {X 76.2263,Y -111.9504,Z 183,A -51.9305,B 4.4543,C 0.3371,E1 4.5577,E2 504.5763} C_DIS
LIN {X 72.3834,Y -114.4721,Z 183,A -53.7496,B 4.4542,C 0.3388,E1 4.5534,E2 506.3809} C_DIS
LIN {X 66.1279,Y -118.1963,Z 183,A -56.7747,B 4.4538,C 0.3429,E1 4.5461,E2 509.4013} C_DIS
LIN {X 62.5002,Y -120.1526,Z 183,A -58.6441,B 4.4535,C 0.3468,E1 4.5415,E2 511.2882} C_DIS
LIN {X 58.9679,Y -121.9256,Z 183,A -60.0205,B 4.4536,C 0.3457,E1 4.5381,E2 512.6279} C_DIS
LIN {X 56.3385,Y -123.1623,Z 183,A -61.26,B 4.4535,C 0.3475,E1 4.535,E2 513.8696} C_DIS
LIN {X 53.6181,Y -124.3696,Z 183,A -62.5786,B 4.4533,C 0.3497,E1 4.5316,E2 515.1967} C_DIS
LIN {X 50.6641,Y -125.6018,Z 183,A -63.8973,B 4.4533,C 0.3509,E1 4.5282,E2 516.5118} C_DIS
LIN {X 47.1092,Y -126.9787,Z 183,A -65.525,B 4.4531,C 0.3529,E1 4.5239,E2 518.1426} C_DIS
LIN {X 42.5843,Y -128.5664,Z 183,A -67.4729,B 4.453,C 0.3541,E1 4.5188,E2 520.0815} C_DIS
LIN {X 39.3413,Y -129.5957,Z 183,A -68.9184,B 4.4529,C 0.3556,E1 4.5149,E2 521.5287} C_DIS
LIN {X 36.2426,Y -130.4962,Z 183,A -70.2052,B 4.4529,C 0.356,E1 4.5115,E2 522.8063} C_DIS
LIN {X 33.1488,Y -131.3161,Z 183,A -71.6314,B 4.4527,C 0.3579,E1 4.5076,E2 524.2427} C_DIS
LIN {X 29.8527,Y -132.1047,Z 183,A -72.9818,B 4.4527,C 0.3581,E1 4.504,E2 525.5833} C_DIS
LIN {X 26.5218,Y -132.8141,Z 183,A -74.4744,B 4.4525,C 0.3597,E1 4.4999,E2 527.0834} C_DIS
LIN {X 21.0519,Y -133.7897,Z 183,A -76.5894,B 4.4526,C 0.3586,E1 4.4941,E2 529.1694} C_DIS
LIN {X 18.2229,Y -134.2054,Z 183,A -78.0808,B 4.4523,C 0.3622,E1 4.4899,E2 530.6979} C_DIS
LIN {X 14.4734,Y -134.6599,Z 183,A -79.9533,B 4.452,C 0.3658,E1 4.4846,E2 532.6065} C_DIS
LIN {X 10.6117,Y -135.0212,Z 183,A -81.4121,B 4.4521,C 0.3645,E1 4.4806,E2 534.0429} C_DIS
LIN {X 4.9407,Y -135.3459,Z 183,A -83.5195,B 4.4523,C 0.3622,E1 4.4748,E2 536.1135} C_DIS
LIN {X 1.5441,Y -135.4287,Z 183,A -85.7018,B 4.4517,C 0.3699,E1 4.4685,E2 538.3919} C_DIS
LIN {X 1.5441,Y -135.4287,Z 183,A -85.7018,B 4.4517,C 0.3699,E1 4.4685,E2 538.3919} C_DIS
Enddeposition()
LIN {X 0.9463,Y -136.3293,Z 183,A -85.9096,B 4.2857,C 0.3677,E1 4.3019,E2 538.6738} C_DIS
Startdeposition()
$VEL.CP = VEL_PRINT
LIN {X 3.8016,Y -136.2837,Z 183,A -82.7605,B 4.2873,C 0.3482,E1 4.3115,E2 535.2706} C_DIS
LIN {X 8.5258,Y -136.0698,Z 183,A -81.6277,B 4.2866,C 0.3563,E1 4.3143,E2 534.2492} C_DIS
LIN {X 15.2913,Y -135.4782,Z 183,A -78.4142,B 4.287,C 0.3515,E1 4.3234,E2 530.9875} C_DIS
LIN {X 18.5784,Y -135.0666,Z 183,A -76.8984,B 4.2872,C 0.3495,E1 4.3276,E2 529.4546} C_DIS
LIN {X 23.8999,Y -134.2253,Z 183,A -74.949,B 4.287,C 0.3514,E1 4.3329,E2 527.5452} C_DIS
LIN {X 26.7986,Y -133.6772,Z 183,A -73.5547,B 4.2872,C 0.349,E1 4.3368,E2 526.1299} C_DIS
LIN {X 30.4579,Y -132.8907,Z 183,A -72.0492,B 4.2872,C 0.3485,E1 4.3408,E2 524.6323} C_DIS
LIN {X 34.6389,Y -131.8636,Z 183,A -70.2777,B 4.2874,C 0.3474,E1 4.3456,E2 522.8646} C_DIS
LIN {X 38.2907,Y -130.8488,Z 183,A -68.7348,B 4.2874,C 0.3465,E1 4.3498,E2 521.3271} C_DIS
LIN {X 41.6095,Y -129.8316,Z 183,A -67.2284,B 4.2876,C 0.3446,E1 4.3538,E2 519.8135} C_DIS
LIN {X 45.6244,Y -128.4773,Z 183,A -65.3956,B 4.2878,C 0.3421,E1 4.3587,E2 517.9728} C_DIS
LIN {X 49.2884,Y -127.115,Z 183,A -63.9991,B 4.2878,C 0.343,E1 4.3622,E2 516.6074} C_DIS
LIN {X 52.2726,Y -125.9175,Z 183,A -62.5498,B 4.2879,C 0.3403,E1 4.366,E2 515.1443} C_DIS
LIN {X 55.0904,Y -124.7116,Z 183,A -61.218,B 4.2881,C 0.3382,E1 4.3694,E2 513.8058} C_DIS
LIN {X 57.6178,Y -123.5634,Z 183,A -59.9786,B 4.2883,C 0.3359,E1 4.3726,E2 512.556} C_DIS
LIN {X 61.1481,Y -121.8567,Z 183,A -58.463,B 4.2883,C 0.3351,E1 4.3764,E2 511.0566} C_DIS
LIN {X 64.8581,Y -119.9235,Z 183,A -56.6931,B 4.2885,C 0.3324,E1 4.3807,E2 509.2839} C_DIS
LIN {X 67.6457,Y -118.373,Z 183,A -54.7372,B 4.2892,C 0.3234,E1 4.3857,E2 507.2459} C_DIS
LIN {X 72.5561,Y -115.4286,Z 183,A -53.0004,B 4.2889,C 0.3273,E1 4.3896,E2 505.5955} C_DIS
LIN {X 76.3341,Y -112.9655,Z 183,A -51.1524,B 4.2891,C 0.3246,E1 4.3939,E2 503.7523} C_DIS
LIN {X 80.1705,Y -110.2761,Z 183,A -49.2539,B 4.2893,C 0.322,E1 4.3982,E2 501.8613} C_DIS
LIN {X 83.7046,Y -107.6182,Z 183,A -47.4139,B 4.2896,C 0.3189,E1 4.4022,E2 500.0222} C_DIS
LIN {X 87.0606,Y -104.9216,Z 183,A -45.6517,B 4.2898,C 0.316,E1 4.4061,E2 498.2648} C_DIS
LIN {X 90.5069,Y -101.964,Z 183,A -43.7629,B 4.29,C 0.3126,E1 4.41,E2 496.377} C_DIS
LIN {X 93.6951,Y -99.0421,Z 183,A -41.9966,B 4.2903,C 0.3095,E1 4.4136,E2 494.6158} C_DIS
LIN {X 96.941,Y -95.8678,Z 183,A -40.1459,B 4.2905,C 0.3063,E1 4.4173,E2 492.771} C_DIS
LIN {X 100.0449,Y -92.6242,Z 183,A -38.2648,B 4.2908,C 0.3023,E1 4.4209,E2 490.889} C_DIS
LIN {X 103.071,Y -89.2445,Z 183,A -36.3938,B 4.291,C 0.2985,E1 4.4243,E2 489.021} C_DIS
LIN {X 106.0252,Y -85.7132,Z 183,A -34.5393,B 4.2913,C 0.2952,E1 4.4276,E2 487.1754} C_DIS
LIN {X 108.8792,Y -82.0574,Z 183,A -32.7435,B 4.2914,C 0.2926,E1 4.4306,E2 485.3979} C_DIS
LIN {X 112.6016,Y -76.8704,Z 183,A -30.2793,B 4.2917,C 0.2889,E1 4.4346,E2 482.9598} C_DIS
LIN {X 116.1732,Y -71.3575,Z 183,A -26.2907,B 4.2931,C 0.2668,E1 4.4407,E2 478.8085} C_DIS
LIN {X 120.2247,Y -64.2976,Z 183,A -23.9749,B 4.2928,C 0.2721,E1 4.4436,E2 476.6344} C_DIS
LIN {X 122.1415,Y -60.5729,Z 183,A -22.4052,B 4.2929,C 0.27,E1 4.4456,E2 475.0879} C_DIS
LIN {X 123.6538,Y -57.4222,Z 183,A -21.1148,B 4.293,C 0.2684,E1 4.4471,E2 473.8193} C_DIS
LIN {X 124.6813,Y -55.1581,Z 183,A -19.7707,B 4.2934,C 0.2619,E1 4.4487,E2 472.4357} C_DIS
LIN {X 126.4255,Y -51.0308,Z 183,A -18.142,B 4.2935,C 0.2601,E1 4.4504,E2 470.8382} C_DIS
LIN {X 127.706,Y -47.7362,Z 183,A -16.654,B 4.2938,C 0.2561,E1 4.4518,E2 469.3488} C_DIS
LIN {X 129.7558,Y -41.8469,Z 183,A -14.1246,B 4.2941,C 0.2502,E1 4.4541,E2 466.829} C_DIS
LIN {X 130.8745,Y -38.2027,Z 183,A -12.6299,B 4.2943,C 0.2471,E1 4.4553,E2 465.3468} C_DIS
LIN {X 131.6756,Y -35.3436,Z 183,A -11.4195,B 4.2945,C 0.2442,E1 4.4562,E2 464.1401} C_DIS
LIN {X 132.4882,Y -32.164,Z 183,A -10.091,B 4.2946,C 0.241,E1 4.4571,E2 462.8171} C_DIS
LIN {X 133.2442,Y -28.872,Z 183,A -8.712,B 4.2948,C 0.2376,E1 4.4579,E2 461.4422} C_DIS
LIN {X 133.9246,Y -25.531,Z 183,A -7.3238,B 4.295,C 0.2341,E1 4.4586,E2 460.0585} C_DIS
LIN {X 134.5039,Y -22.2789,Z 183,A -6.0166,B 4.2952,C 0.2313,E1 4.4593,E2 458.7606} C_DIS
LIN {X 135.0746,Y -18.5227,Z 183,A -4.4255,B 4.2954,C 0.2269,E1 4.4599,E2 457.1691} C_DIS
LIN {X 135.6915,Y -13.2484,Z 183,A -1.9178,B 4.2959,C 0.217,E1 4.4607,E2 454.6243} C_DIS
LIN {X 135.9978,Y -9.6101,Z 183,A -0.7142,B 4.2959,C 0.217,E1 4.4609,E2 453.4619} C_DIS
Enddeposition()
END
